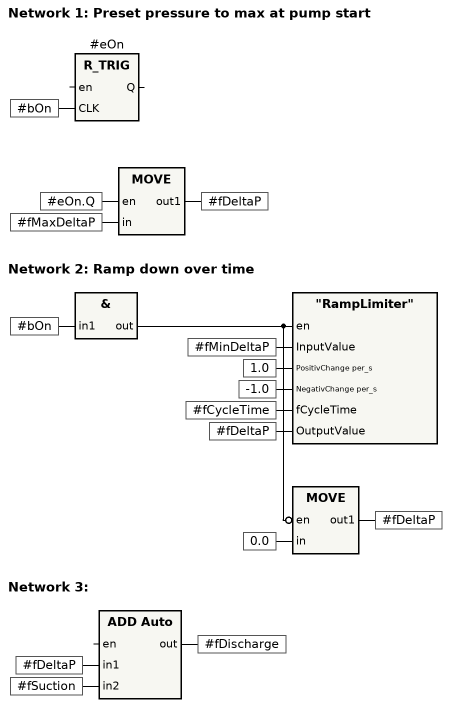
   #eOn(CLK := #bOn);   // R_TRIG
   IF #eOn.Q THEN #fDeltaP := #fMaxDeltaP; END_IF;
END_REGION

REGION Network 2: Ramp down over time
   // When pump is off, delta P is zero.
   // When the pump runs, it starts at the max pressure and ramps down to the min pressure to approximate the decrease in liquid on the suction side
   IF #bOn THEN
       "RampLimiter"(InputValue := #fMinDeltaP,
                     "PositivChange per_s" := 1.0,
                     "NegativChange per_s" := -1.0,
                     fCycleTime := #fCycleTime,
                     OutputValue := #fDeltaP);
   END_IF;
   IF NOT #bOn THEN #fDeltaP := 0.0; END_IF;
END_REGION

REGION Network 3
   #fDischarge := #fDeltaP + #fSuction;
END_REGION
END_FUNCTION_BLOCK

FUNCTION "RampLimiter" : Void
{ S7_Optimized_Access := 'TRUE' }
VERSION : 0.1
   VAR_INPUT 
      InputValue : Real;
      "PositivChange per_s" : Real;
      "NegativChange per_s" : Real;
      fCycleTime : Real;
   END_VAR

   VAR_IN_OUT 
      OutputValue : Real;
   END_VAR


BEGIN
	#OutputValue += MAX(IN1:=MIN(IN1:=#InputValue-#OutputValue,IN2:=#"PositivChange per_s"*#fCycleTime),IN2:=#"NegativChange per_s"*#fCycleTime);
END_FUNCTION

FUNCTION_BLOCK "InputAlarmHandling"   // FB38, FBD
TITLE = Handle I/O alarms
{ S7_Optimized_Access := 'TRUE' }
AUTHOR : Heaten
VERSION : 0.1
// Handle I/O alarms
// stored: AutoNumber true, IsIECCheckEnabled false, IsRetainMemResEnabled false, MemoryReserve 0, SetENOAutomatically false, UDAEnableTagReadback false
   VAR
      A1102 { ExternalAccessible := 'False'; ExternalVisible := 'False'; ExternalWritable := 'False'; S7_SetPoint := 'True'} : "fbDigitalAlarm";
      A1103 { S7_SetPoint := 'True'} : "fbDigitalAlarm";
      A1110 { ExternalAccessible := 'False'; ExternalVisible := 'False'; ExternalWritable := 'False'; S7_SetPoint := 'True'} : "fbDigitalAlarm";
      A1122 { ExternalAccessible := 'False'; ExternalVisible := 'False'; ExternalWritable := 'False'; S7_SetPoint := 'True'} : "fbDigitalAlarm";
      A1123 { S7_SetPoint := 'True'} : "fbDigitalAlarm";
      A1130 { ExternalAccessible := 'False'; ExternalVisible := 'False'; ExternalWritable := 'False'; S7_SetPoint := 'True'} : "fbDigitalAlarm";
      A1142 { ExternalAccessible := 'False'; ExternalVisible := 'False'; ExternalWritable := 'False'; S7_SetPoint := 'True'} : "fbDigitalAlarm";
      A1143 { S7_SetPoint := 'True'} : "fbDigitalAlarm";
      A1150 { ExternalAccessible := 'False'; ExternalVisible := 'False'; ExternalWritable := 'False'; S7_SetPoint := 'True'} : "fbDigitalAlarm";
      A1201 { ExternalAccessible := 'False'; ExternalVisible := 'False'; ExternalWritable := 'False'; S7_SetPoint := 'True'} : "fbHMIEvent";
      A1202 { ExternalAccessible := 'False'; ExternalVisible := 'False'; ExternalWritable := 'False'; S7_SetPoint := 'True'} : "fbHMIEvent";
      A1203 { ExternalAccessible := 'False'; ExternalVisible := 'False'; ExternalWritable := 'False'; S7_SetPoint := 'True'} : "fbHMIEvent";
      A1204 { ExternalAccessible := 'False'; ExternalVisible := 'False'; ExternalWritable := 'False'; S7_SetPoint := 'True'} : "fbHMIEvent";
      A1205 { ExternalAccessible := 'False'; ExternalVisible := 'False'; ExternalWritable := 'False'; S7_SetPoint := 'True'} : "fbHMIEvent";
      A1206 { ExternalAccessible := 'False'; ExternalVisible := 'False'; ExternalWritable := 'False'; S7_SetPoint := 'True'} : "fbHMIEvent";
      A1207 { ExternalAccessible := 'False'; ExternalVisible := 'False'; ExternalWritable := 'False'; S7_SetPoint := 'True'} : "fbHMIEvent";
      A1208 { ExternalAccessible := 'False'; ExternalVisible := 'False'; ExternalWritable := 'False'; S7_SetPoint := 'True'} : "fbHMIEvent";
      A1209 { ExternalAccessible := 'False'; ExternalVisible := 'False'; ExternalWritable := 'False'; S7_SetPoint := 'True'} : "fbHMIEvent";
      A1210 { ExternalAccessible := 'False'; ExternalVisible := 'False'; ExternalWritable := 'False'; S7_SetPoint := 'True'} : "fbHMIEvent";
      A1212 { ExternalAccessible := 'False'; ExternalVisible := 'False'; ExternalWritable := 'False'; S7_SetPoint := 'True'} : "fbHMIEvent";
      A1213 { ExternalAccessible := 'False'; ExternalVisible := 'False'; ExternalWritable := 'False'; S7_SetPoint := 'True'} : "fbHMIEvent";
      A1214 { ExternalAccessible := 'False'; ExternalVisible := 'False'; ExternalWritable := 'False'; S7_SetPoint := 'True'} : "fbHMIEvent";
      A1215 { ExternalAccessible := 'False'; ExternalVisible := 'False'; ExternalWritable := 'False'; S7_SetPoint := 'True'} : "fbHMIEvent";
      A1220 { ExternalAccessible := 'False'; ExternalVisible := 'False'; ExternalWritable := 'False'; S7_SetPoint := 'True'} : "fbHMIEvent";
      A1221 { ExternalAccessible := 'False'; ExternalVisible := 'False'; ExternalWritable := 'False'; S7_SetPoint := 'True'} : "fbHMIEvent";
      A1223 { ExternalAccessible := 'False'; ExternalVisible := 'False'; ExternalWritable := 'False'; S7_SetPoint := 'True'} : "fbHMIEvent";
      A1231 { ExternalAccessible := 'False'; ExternalVisible := 'False'; ExternalWritable := 'False'; S7_SetPoint := 'True'} : "fbHMIEvent";
      A1232 { ExternalAccessible := 'False'; ExternalVisible := 'False'; ExternalWritable := 'False'; S7_SetPoint := 'True'} : "fbHMIEvent";
      A1233 { ExternalAccessible := 'False'; ExternalVisible := 'False'; ExternalWritable := 'False'; S7_SetPoint := 'True'} : "fbDigitalAlarm";
      A1241 { ExternalAccessible := 'False'; ExternalVisible := 'False'; ExternalWritable := 'False'; S7_SetPoint := 'True'} : "fbHMIEvent";
      A1242 { ExternalAccessible := 'False'; ExternalVisible := 'False'; ExternalWritable := 'False'; S7_SetPoint := 'True'} : "fbHMIEvent";
      A1243 { ExternalAccessible := 'False'; ExternalVisible := 'False'; ExternalWritable := 'False'; S7_SetPoint := 'True'} : "fbHMIEvent";
      A1244 { ExternalAccessible := 'False'; ExternalVisible := 'False'; ExternalWritable := 'False'; S7_SetPoint := 'True'} : "fbHMIEvent";
      A1255 { ExternalAccessible := 'False'; ExternalVisible := 'False'; ExternalWritable := 'False'; S7_SetPoint := 'True'} : "fbHMIEvent";
      A1256 { ExternalAccessible := 'False'; ExternalVisible := 'False'; ExternalWritable := 'False'; S7_SetPoint := 'True'} : "fbHMIEvent";
      A1257 { ExternalAccessible := 'False'; ExternalVisible := 'False'; ExternalWritable := 'False'; S7_SetPoint := 'True'} : "fbHMIEvent";
      A1264 { ExternalAccessible := 'False'; ExternalVisible := 'False'; ExternalWritable := 'False'; S7_SetPoint := 'True'} : "fbHMIEvent";
      A1266 { ExternalAccessible := 'False'; ExternalVisible := 'False'; ExternalWritable := 'False'; S7_SetPoint := 'True'} : "fbHMIEvent";
      A1267 { ExternalAccessible := 'False'; ExternalVisible := 'False'; ExternalWritable := 'False'; S7_SetPoint := 'True'} : "fbHMIEvent";
      A1268 { ExternalAccessible := 'False'; ExternalVisible := 'False'; ExternalWritable := 'False'; S7_SetPoint := 'True'} : "fbHMIEvent";
      A1274 { S7_SetPoint := 'True'} : "fbHMIEvent";
      A1276 { S7_SetPoint := 'True'} : "fbHMIEvent";
      A1277 { S7_SetPoint := 'True'} : "fbHMIEvent";
      A1278 { S7_SetPoint := 'True'} : "fbHMIEvent";
      A1279 { S7_SetPoint := 'True'} : "fbHMIEvent";
      A1280 { S7_SetPoint := 'True'} : "fbHMIEvent";
      A1281 { S7_SetPoint := 'True'} : "fbHMIEvent";
      A1282 { S7_SetPoint := 'True'} : "fbHMIEvent";
      A1283 { S7_SetPoint := 'True'} : "fbHMIEvent";
      A1284 { S7_SetPoint := 'True'} : "fbHMIEvent";
      A1285 { S7_SetPoint := 'True'} : "fbHMIEvent";
      A1286 { S7_SetPoint := 'True'} : "fbHMIEvent";
      A1287 { S7_SetPoint := 'True'} : "fbHMIEvent";
      A1288 { S7_SetPoint := 'True'} : "fbHMIEvent";
      A1289 { S7_SetPoint := 'True'} : "fbHMIEvent";
      A1290 { S7_SetPoint := 'True'} : "fbHMIEvent";
      A1291 { S7_SetPoint := 'True'} : "fbHMIEvent";
      A1292 { S7_SetPoint := 'True'} : "fbHMIEvent";
      A5250 { ExternalAccessible := 'False'; ExternalVisible := 'False'; ExternalWritable := 'False'; S7_SetPoint := 'True'} : "fbHMIEvent";
      A5251 { ExternalAccessible := 'False'; ExternalVisible := 'False'; ExternalWritable := 'False'; S7_SetPoint := 'True'} : "fbHMIEvent";
      A5252 { ExternalAccessible := 'False'; ExternalVisible := 'False'; ExternalWritable := 'False'; S7_SetPoint := 'True'} : "fbHMIEvent";
      A5253 { ExternalAccessible := 'False'; ExternalVisible := 'False'; ExternalWritable := 'False'; S7_SetPoint := 'True'} : "fbHMIEvent";
      A5254 { ExternalAccessible := 'False'; ExternalVisible := 'False'; ExternalWritable := 'False'; S7_SetPoint := 'True'} : "fbHMIEvent";
      A5255 { ExternalAccessible := 'False'; ExternalVisible := 'False'; ExternalWritable := 'False'; S7_SetPoint := 'True'} : "fbHMIEvent";
   END_VAR
BEGIN

REGION Network 1: 1102
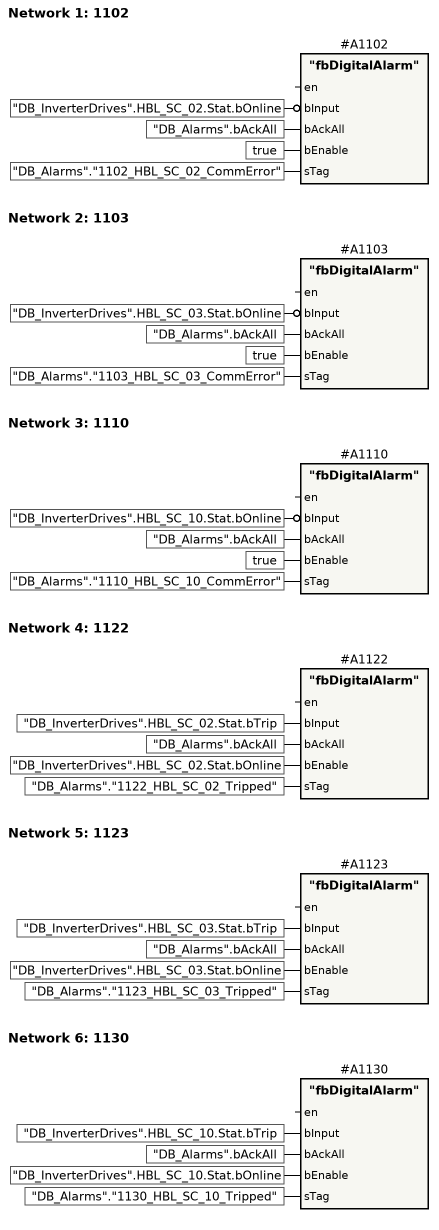
   #A1102(bInput := NOT "DB_InverterDrives".HBL_SC_02.Stat.bOnline,   // "fbDigitalAlarm"
          bAckAll := "DB_Alarms".bAckAll,
          bEnable := true,
          sTag := "DB_Alarms"."1102_HBL_SC_02_CommError");
END_REGION

REGION Network 2: 1103
   #A1103(bInput := NOT "DB_InverterDrives".HBL_SC_03.Stat.bOnline,   // "fbDigitalAlarm"
          bAckAll := "DB_Alarms".bAckAll,
          bEnable := true,
          sTag := "DB_Alarms"."1103_HBL_SC_03_CommError");
END_REGION

REGION Network 3: 1110
   #A1110(bInput := NOT "DB_InverterDrives".HBL_SC_10.Stat.bOnline,   // "fbDigitalAlarm"
          bAckAll := "DB_Alarms".bAckAll,
          bEnable := true,
          sTag := "DB_Alarms"."1110_HBL_SC_10_CommError");
END_REGION

REGION Network 4: 1122
   // Only show if online
   #A1122(bInput := "DB_InverterDrives".HBL_SC_02.Stat.bTrip,   // "fbDigitalAlarm"
          bAckAll := "DB_Alarms".bAckAll,
          bEnable := "DB_InverterDrives".HBL_SC_02.Stat.bOnline,
          sTag := "DB_Alarms"."1122_HBL_SC_02_Tripped");
END_REGION

REGION Network 5: 1123
   // Only show if online
   #A1123(bInput := "DB_InverterDrives".HBL_SC_03.Stat.bTrip,   // "fbDigitalAlarm"
          bAckAll := "DB_Alarms".bAckAll,
          bEnable := "DB_InverterDrives".HBL_SC_03.Stat.bOnline,
          sTag := "DB_Alarms"."1123_HBL_SC_03_Tripped");
END_REGION

REGION Network 6: 1130
   // Only show if online
   #A1130(bInput := "DB_InverterDrives".HBL_SC_10.Stat.bTrip,   // "fbDigitalAlarm"
          bAckAll := "DB_Alarms".bAckAll,
          bEnable := "DB_InverterDrives".HBL_SC_10.Stat.bOnline,
          sTag := "DB_Alarms"."1130_HBL_SC_10_Tripped");
END_REGION

REGION Network 7: 1142
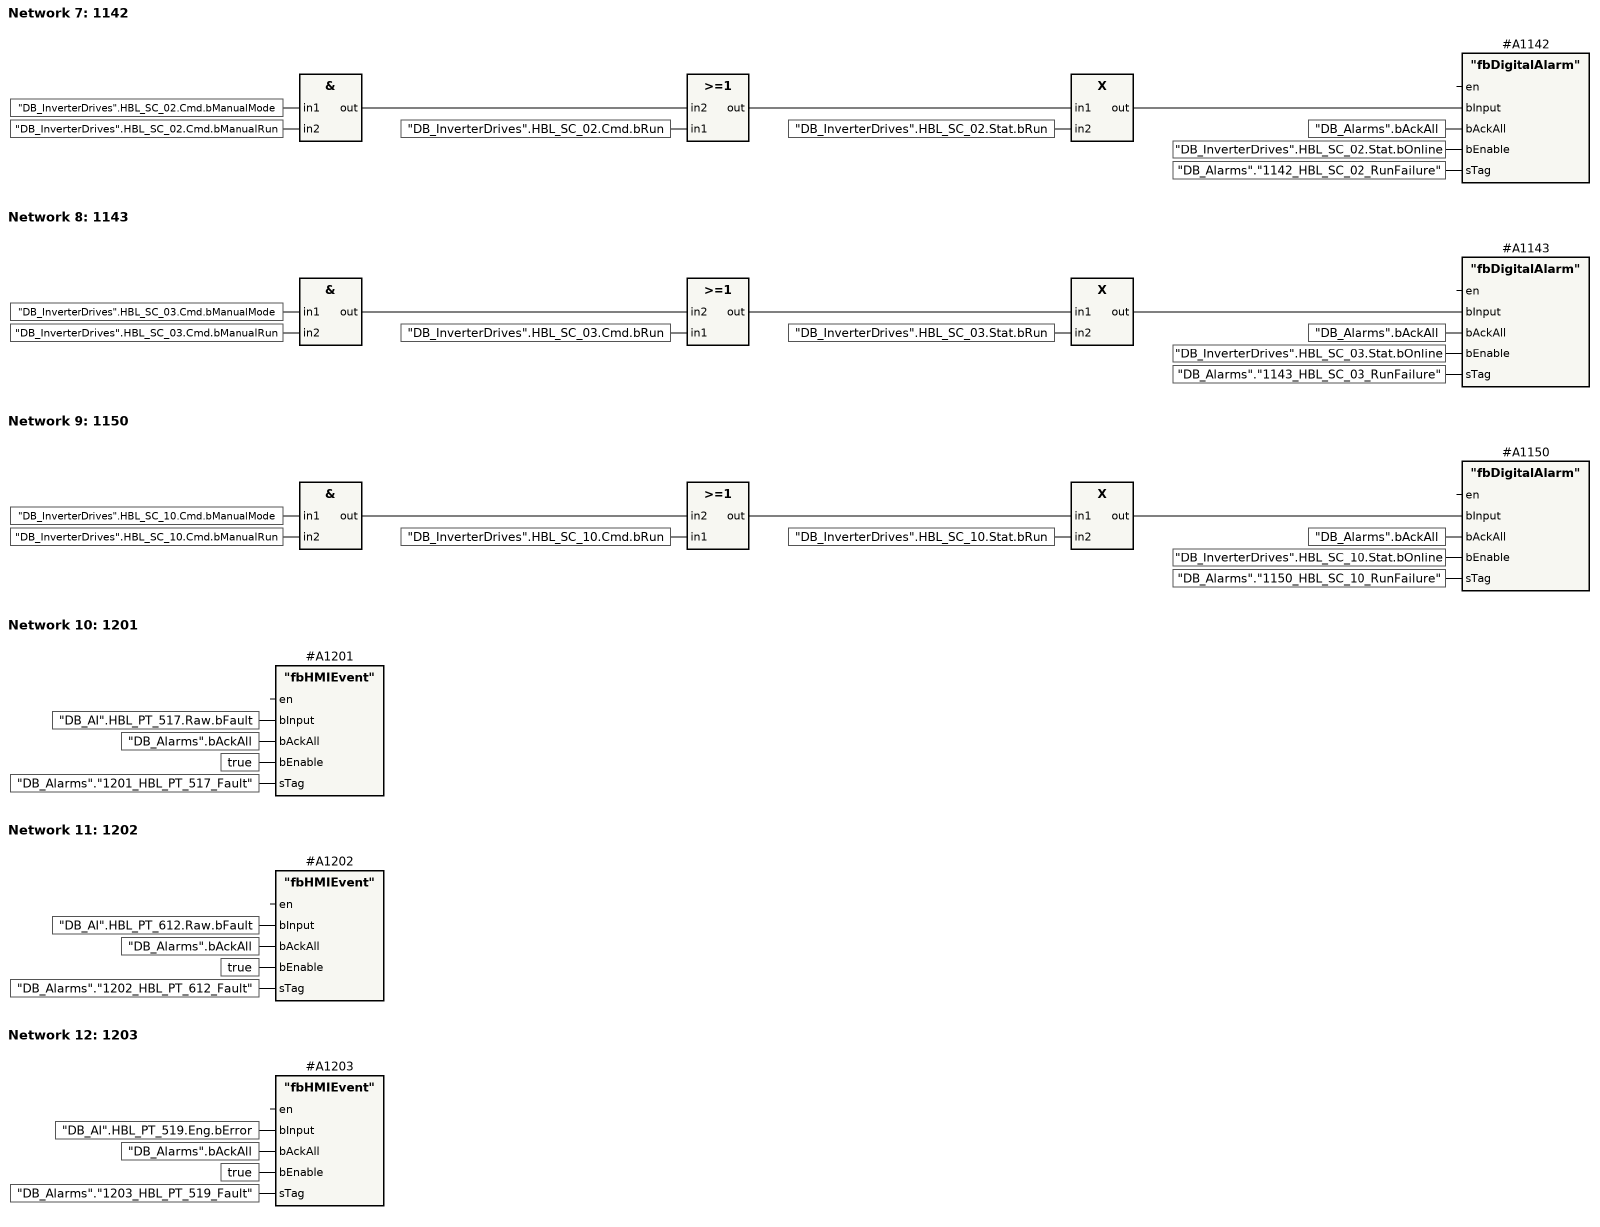
   #A1142(bInput := (("DB_InverterDrives".HBL_SC_02.Cmd.bManualMode AND "DB_InverterDrives".HBL_SC_02.Cmd.bManualRun) OR "DB_InverterDrives".HBL_SC_02.Cmd.bRun) XOR "DB_InverterDrives".HBL_SC_02.Stat.bRun,   // "fbDigitalAlarm"
          bAckAll := "DB_Alarms".bAckAll,
          bEnable := "DB_InverterDrives".HBL_SC_02.Stat.bOnline,
          sTag := "DB_Alarms"."1142_HBL_SC_02_RunFailure");
END_REGION

REGION Network 8: 1143
   #A1143(bInput := (("DB_InverterDrives".HBL_SC_03.Cmd.bManualMode AND "DB_InverterDrives".HBL_SC_03.Cmd.bManualRun) OR "DB_InverterDrives".HBL_SC_03.Cmd.bRun) XOR "DB_InverterDrives".HBL_SC_03.Stat.bRun,   // "fbDigitalAlarm"
          bAckAll := "DB_Alarms".bAckAll,
          bEnable := "DB_InverterDrives".HBL_SC_03.Stat.bOnline,
          sTag := "DB_Alarms"."1143_HBL_SC_03_RunFailure");
END_REGION

REGION Network 9: 1150
   #A1150(bInput := (("DB_InverterDrives".HBL_SC_10.Cmd.bManualMode AND "DB_InverterDrives".HBL_SC_10.Cmd.bManualRun) OR "DB_InverterDrives".HBL_SC_10.Cmd.bRun) XOR "DB_InverterDrives".HBL_SC_10.Stat.bRun,   // "fbDigitalAlarm"
          bAckAll := "DB_Alarms".bAckAll,
          bEnable := "DB_InverterDrives".HBL_SC_10.Stat.bOnline,
          sTag := "DB_Alarms"."1150_HBL_SC_10_RunFailure");
END_REGION

REGION Network 10: 1201
   #A1201(bInput := "DB_AI".HBL_PT_517.Raw.bFault,   // "fbHMIEvent"
          bAckAll := "DB_Alarms".bAckAll,
          bEnable := true,
          sTag := "DB_Alarms"."1201_HBL_PT_517_Fault");
END_REGION

REGION Network 11: 1202
   #A1202(bInput := "DB_AI".HBL_PT_612.Raw.bFault,   // "fbHMIEvent"
          bAckAll := "DB_Alarms".bAckAll,
          bEnable := true,
          sTag := "DB_Alarms"."1202_HBL_PT_612_Fault");
END_REGION

REGION Network 12: 1203
   #A1203(bInput := "DB_AI".HBL_PT_519.Eng.bError,   // "fbHMIEvent"
          bAckAll := "DB_Alarms".bAckAll,
          bEnable := true,
          sTag := "DB_Alarms"."1203_HBL_PT_519_Fault");
END_REGION

REGION Network 13: 1204
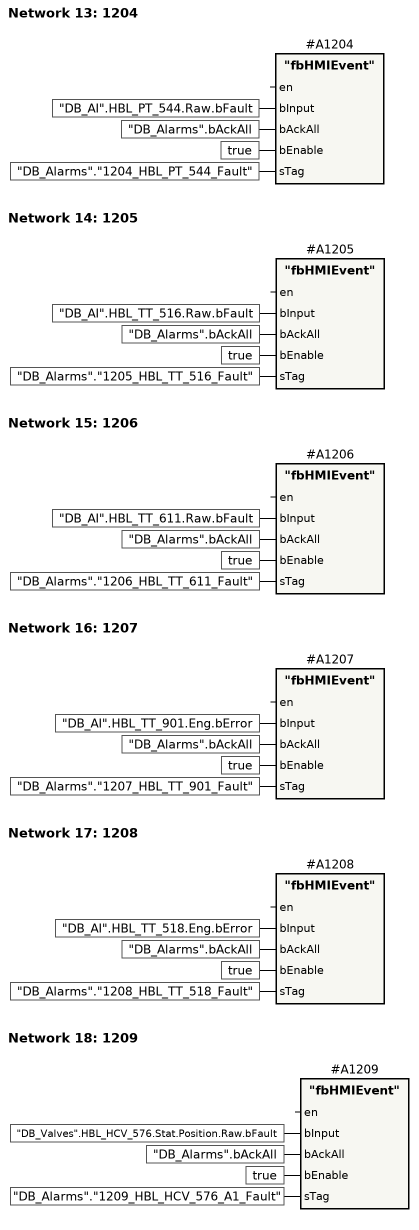
   #A1204(bInput := "DB_AI".HBL_PT_544.Raw.bFault,   // "fbHMIEvent"
          bAckAll := "DB_Alarms".bAckAll,
          bEnable := true,
          sTag := "DB_Alarms"."1204_HBL_PT_544_Fault");
END_REGION

REGION Network 14: 1205
   #A1205(bInput := "DB_AI".HBL_TT_516.Raw.bFault,   // "fbHMIEvent"
          bAckAll := "DB_Alarms".bAckAll,
          bEnable := true,
          sTag := "DB_Alarms"."1205_HBL_TT_516_Fault");
END_REGION

REGION Network 15: 1206
   #A1206(bInput := "DB_AI".HBL_TT_611.Raw.bFault,   // "fbHMIEvent"
          bAckAll := "DB_Alarms".bAckAll,
          bEnable := true,
          sTag := "DB_Alarms"."1206_HBL_TT_611_Fault");
END_REGION

REGION Network 16: 1207
   #A1207(bInput := "DB_AI".HBL_TT_901.Eng.bError,   // "fbHMIEvent"
          bAckAll := "DB_Alarms".bAckAll,
          bEnable := true,
          sTag := "DB_Alarms"."1207_HBL_TT_901_Fault");
END_REGION

REGION Network 17: 1208
   #A1208(bInput := "DB_AI".HBL_TT_518.Eng.bError,   // "fbHMIEvent"
          bAckAll := "DB_Alarms".bAckAll,
          bEnable := true,
          sTag := "DB_Alarms"."1208_HBL_TT_518_Fault");
END_REGION

REGION Network 18: 1209
   #A1209(bInput := "DB_Valves".HBL_HCV_576.Stat.Position.Raw.bFault,   // "fbHMIEvent"
          bAckAll := "DB_Alarms".bAckAll,
          bEnable := true,
          sTag := "DB_Alarms"."1209_HBL_HCV_576_A1_Fault");
END_REGION

REGION Network 19: 1210
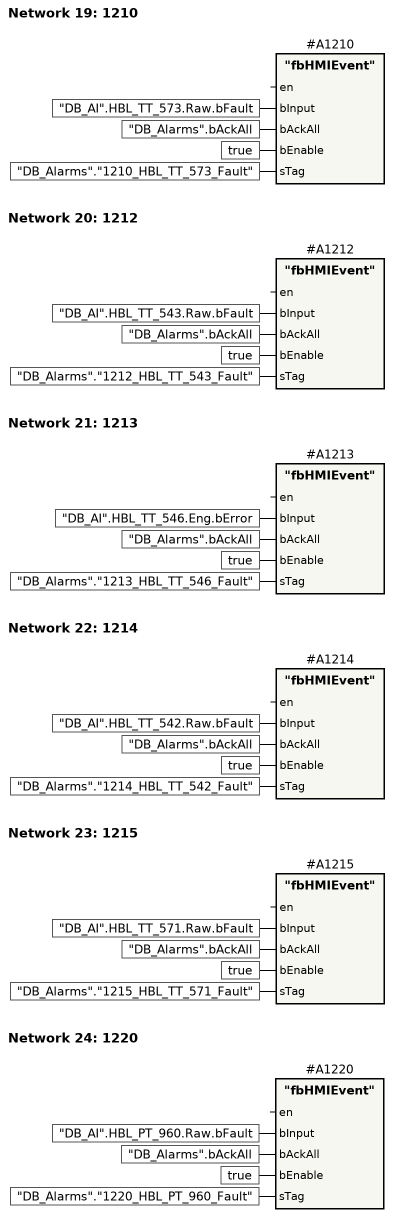
   #A1210(bInput := "DB_AI".HBL_TT_573.Raw.bFault,   // "fbHMIEvent"
          bAckAll := "DB_Alarms".bAckAll,
          bEnable := true,
          sTag := "DB_Alarms"."1210_HBL_TT_573_Fault");
END_REGION

REGION Network 20: 1212
   #A1212(bInput := "DB_AI".HBL_TT_543.Raw.bFault,   // "fbHMIEvent"
          bAckAll := "DB_Alarms".bAckAll,
          bEnable := true,
          sTag := "DB_Alarms"."1212_HBL_TT_543_Fault");
END_REGION

REGION Network 21: 1213
   #A1213(bInput := "DB_AI".HBL_TT_546.Eng.bError,   // "fbHMIEvent"
          bAckAll := "DB_Alarms".bAckAll,
          bEnable := true,
          sTag := "DB_Alarms"."1213_HBL_TT_546_Fault");
END_REGION

REGION Network 22: 1214
   #A1214(bInput := "DB_AI".HBL_TT_542.Raw.bFault,   // "fbHMIEvent"
          bAckAll := "DB_Alarms".bAckAll,
          bEnable := true,
          sTag := "DB_Alarms"."1214_HBL_TT_542_Fault");
END_REGION

REGION Network 23: 1215
   #A1215(bInput := "DB_AI".HBL_TT_571.Raw.bFault,   // "fbHMIEvent"
          bAckAll := "DB_Alarms".bAckAll,
          bEnable := true,
          sTag := "DB_Alarms"."1215_HBL_TT_571_Fault");
END_REGION

REGION Network 24: 1220
   #A1220(bInput := "DB_AI".HBL_PT_960.Raw.bFault,   // "fbHMIEvent"
          bAckAll := "DB_Alarms".bAckAll,
          bEnable := true,
          sTag := "DB_Alarms"."1220_HBL_PT_960_Fault");
END_REGION

REGION Network 25: 1221
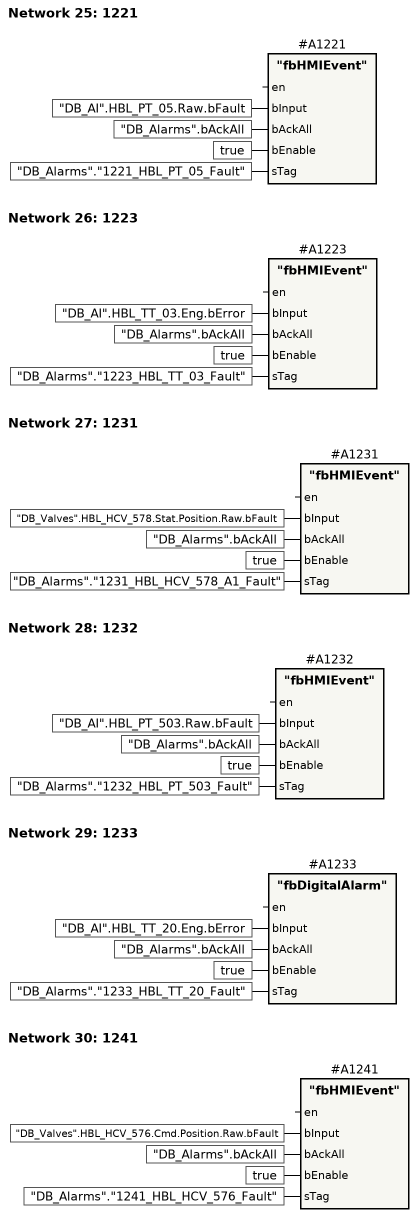
   #A1221(bInput := "DB_AI".HBL_PT_05.Raw.bFault,   // "fbHMIEvent"
          bAckAll := "DB_Alarms".bAckAll,
          bEnable := true,
          sTag := "DB_Alarms"."1221_HBL_PT_05_Fault");
END_REGION

REGION Network 26: 1223
   #A1223(bInput := "DB_AI".HBL_TT_03.Eng.bError,   // "fbHMIEvent"
          bAckAll := "DB_Alarms".bAckAll,
          bEnable := true,
          sTag := "DB_Alarms"."1223_HBL_TT_03_Fault");
END_REGION

REGION Network 27: 1231
   #A1231(bInput := "DB_Valves".HBL_HCV_578.Stat.Position.Raw.bFault,   // "fbHMIEvent"
          bAckAll := "DB_Alarms".bAckAll,
          bEnable := true,
          sTag := "DB_Alarms"."1231_HBL_HCV_578_A1_Fault");
END_REGION

REGION Network 28: 1232
   #A1232(bInput := "DB_AI".HBL_PT_503.Raw.bFault,   // "fbHMIEvent"
          bAckAll := "DB_Alarms".bAckAll,
          bEnable := true,
          sTag := "DB_Alarms"."1232_HBL_PT_503_Fault");
END_REGION

REGION Network 29: 1233
   #A1233(bInput := "DB_AI".HBL_TT_20.Eng.bError,   // "fbDigitalAlarm"
          bAckAll := "DB_Alarms".bAckAll,
          bEnable := true,
          sTag := "DB_Alarms"."1233_HBL_TT_20_Fault");
END_REGION

REGION Network 30: 1241
   #A1241(bInput := "DB_Valves".HBL_HCV_576.Cmd.Position.Raw.bFault,   // "fbHMIEvent"
          bAckAll := "DB_Alarms".bAckAll,
          bEnable := true,
          sTag := "DB_Alarms"."1241_HBL_HCV_576_Fault");
END_REGION

REGION Network 31: 1242
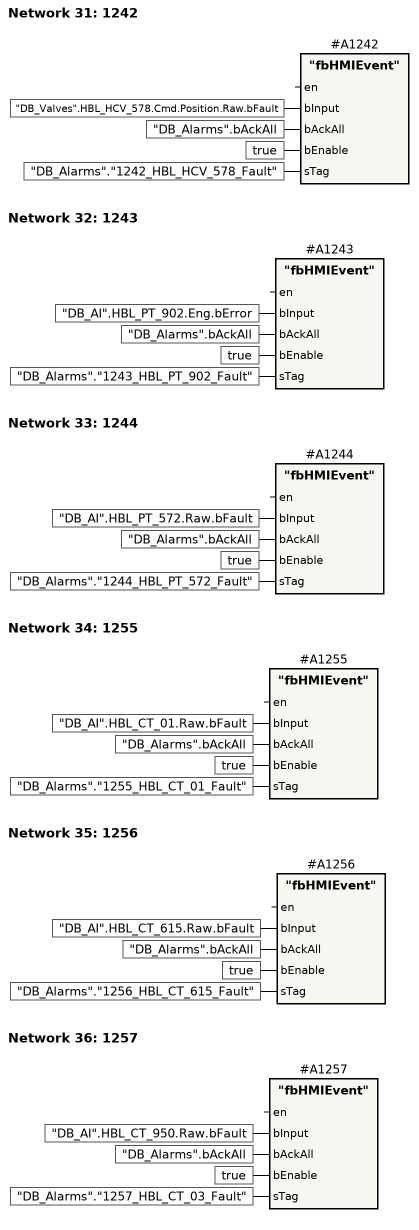
   #A1242(bInput := "DB_Valves".HBL_HCV_578.Cmd.Position.Raw.bFault,   // "fbHMIEvent"
          bAckAll := "DB_Alarms".bAckAll,
          bEnable := true,
          sTag := "DB_Alarms"."1242_HBL_HCV_578_Fault");
END_REGION

REGION Network 32: 1243
   #A1243(bInput := "DB_AI".HBL_PT_902.Eng.bError,   // "fbHMIEvent"
          bAckAll := "DB_Alarms".bAckAll,
          bEnable := true,
          sTag := "DB_Alarms"."1243_HBL_PT_902_Fault");
END_REGION

REGION Network 33: 1244
   #A1244(bInput := "DB_AI".HBL_PT_572.Raw.bFault,   // "fbHMIEvent"
          bAckAll := "DB_Alarms".bAckAll,
          bEnable := true,
          sTag := "DB_Alarms"."1244_HBL_PT_572_Fault");
END_REGION

REGION Network 34: 1255
   #A1255(bInput := "DB_AI".HBL_CT_01.Raw.bFault,   // "fbHMIEvent"
          bAckAll := "DB_Alarms".bAckAll,
          bEnable := true,
          sTag := "DB_Alarms"."1255_HBL_CT_01_Fault");
END_REGION

REGION Network 35: 1256
   #A1256(bInput := "DB_AI".HBL_CT_615.Raw.bFault,   // "fbHMIEvent"
          bAckAll := "DB_Alarms".bAckAll,
          bEnable := true,
          sTag := "DB_Alarms"."1256_HBL_CT_615_Fault");
END_REGION

REGION Network 36: 1257
   #A1257(bInput := "DB_AI".HBL_CT_950.Raw.bFault,   // "fbHMIEvent"
          bAckAll := "DB_Alarms".bAckAll,
          bEnable := true,
          sTag := "DB_Alarms"."1257_HBL_CT_03_Fault");
END_REGION

REGION Network 37: 1264
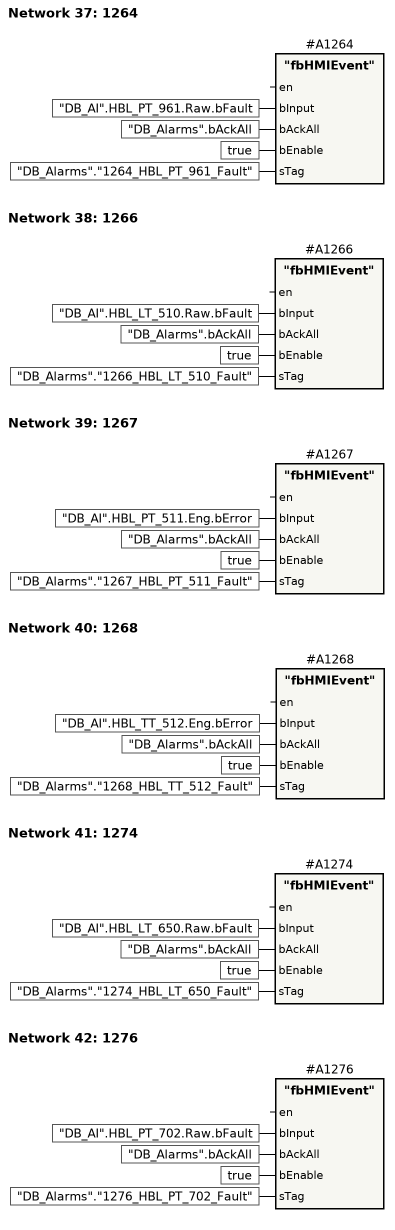
   #A1264(bInput := "DB_AI".HBL_PT_961.Raw.bFault,   // "fbHMIEvent"
          bAckAll := "DB_Alarms".bAckAll,
          bEnable := true,
          sTag := "DB_Alarms"."1264_HBL_PT_961_Fault");
END_REGION

REGION Network 38: 1266
   #A1266(bInput := "DB_AI".HBL_LT_510.Raw.bFault,   // "fbHMIEvent"
          bAckAll := "DB_Alarms".bAckAll,
          bEnable := true,
          sTag := "DB_Alarms"."1266_HBL_LT_510_Fault");
END_REGION

REGION Network 39: 1267
   #A1267(bInput := "DB_AI".HBL_PT_511.Eng.bError,   // "fbHMIEvent"
          bAckAll := "DB_Alarms".bAckAll,
          bEnable := true,
          sTag := "DB_Alarms"."1267_HBL_PT_511_Fault");
END_REGION

REGION Network 40: 1268
   #A1268(bInput := "DB_AI".HBL_TT_512.Eng.bError,   // "fbHMIEvent"
          bAckAll := "DB_Alarms".bAckAll,
          bEnable := true,
          sTag := "DB_Alarms"."1268_HBL_TT_512_Fault");
END_REGION

REGION Network 41: 1274
   #A1274(bInput := "DB_AI".HBL_LT_650.Raw.bFault,   // "fbHMIEvent"
          bAckAll := "DB_Alarms".bAckAll,
          bEnable := true,
          sTag := "DB_Alarms"."1274_HBL_LT_650_Fault");
END_REGION

REGION Network 42: 1276
   #A1276(bInput := "DB_AI".HBL_PT_702.Raw.bFault,   // "fbHMIEvent"
          bAckAll := "DB_Alarms".bAckAll,
          bEnable := true,
          sTag := "DB_Alarms"."1276_HBL_PT_702_Fault");
END_REGION

REGION Network 43: 1277
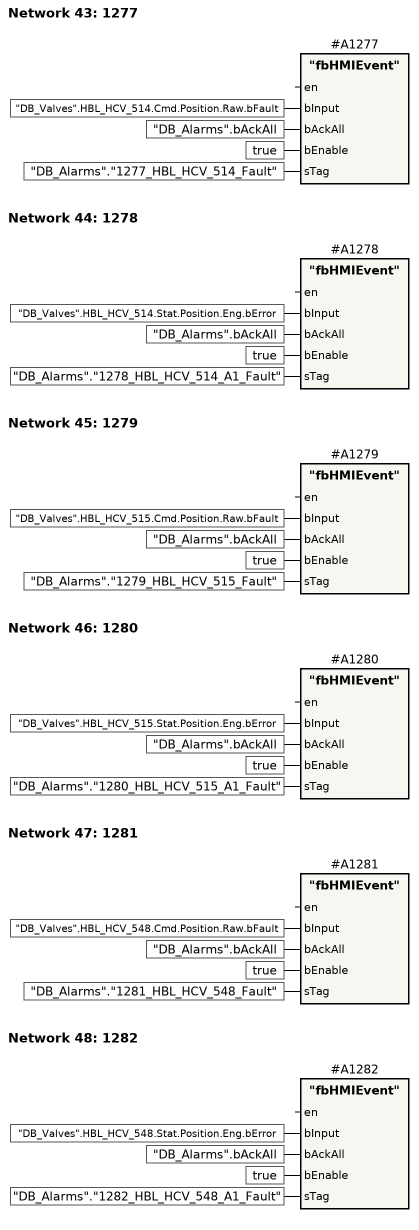
   #A1277(bInput := "DB_Valves".HBL_HCV_514.Cmd.Position.Raw.bFault,   // "fbHMIEvent"
          bAckAll := "DB_Alarms".bAckAll,
          bEnable := true,
          sTag := "DB_Alarms"."1277_HBL_HCV_514_Fault");
END_REGION

REGION Network 44: 1278
   #A1278(bInput := "DB_Valves".HBL_HCV_514.Stat.Position.Eng.bError,   // "fbHMIEvent"
          bAckAll := "DB_Alarms".bAckAll,
          bEnable := true,
          sTag := "DB_Alarms"."1278_HBL_HCV_514_A1_Fault");
END_REGION

REGION Network 45: 1279
   #A1279(bInput := "DB_Valves".HBL_HCV_515.Cmd.Position.Raw.bFault,   // "fbHMIEvent"
          bAckAll := "DB_Alarms".bAckAll,
          bEnable := true,
          sTag := "DB_Alarms"."1279_HBL_HCV_515_Fault");
END_REGION

REGION Network 46: 1280
   #A1280(bInput := "DB_Valves".HBL_HCV_515.Stat.Position.Eng.bError,   // "fbHMIEvent"
          bAckAll := "DB_Alarms".bAckAll,
          bEnable := true,
          sTag := "DB_Alarms"."1280_HBL_HCV_515_A1_Fault");
END_REGION

REGION Network 47: 1281
   #A1281(bInput := "DB_Valves".HBL_HCV_548.Cmd.Position.Raw.bFault,   // "fbHMIEvent"
          bAckAll := "DB_Alarms".bAckAll,
          bEnable := true,
          sTag := "DB_Alarms"."1281_HBL_HCV_548_Fault");
END_REGION

REGION Network 48: 1282
   #A1282(bInput := "DB_Valves".HBL_HCV_548.Stat.Position.Eng.bError,   // "fbHMIEvent"
          bAckAll := "DB_Alarms".bAckAll,
          bEnable := true,
          sTag := "DB_Alarms"."1282_HBL_HCV_548_A1_Fault");
END_REGION

REGION Network 49: 1283
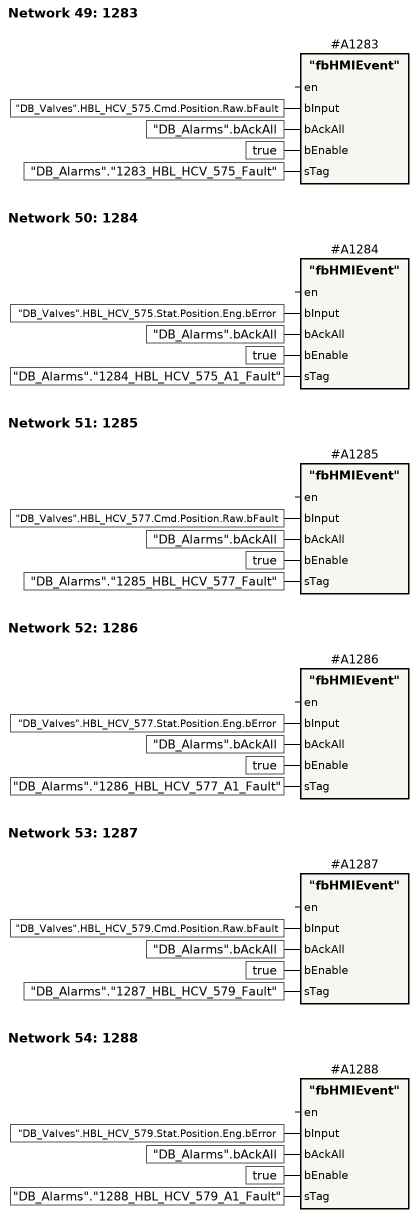
   #A1283(bInput := "DB_Valves".HBL_HCV_575.Cmd.Position.Raw.bFault,   // "fbHMIEvent"
          bAckAll := "DB_Alarms".bAckAll,
          bEnable := true,
          sTag := "DB_Alarms"."1283_HBL_HCV_575_Fault");
END_REGION

REGION Network 50: 1284
   #A1284(bInput := "DB_Valves".HBL_HCV_575.Stat.Position.Eng.bError,   // "fbHMIEvent"
          bAckAll := "DB_Alarms".bAckAll,
          bEnable := true,
          sTag := "DB_Alarms"."1284_HBL_HCV_575_A1_Fault");
END_REGION

REGION Network 51: 1285
   #A1285(bInput := "DB_Valves".HBL_HCV_577.Cmd.Position.Raw.bFault,   // "fbHMIEvent"
          bAckAll := "DB_Alarms".bAckAll,
          bEnable := true,
          sTag := "DB_Alarms"."1285_HBL_HCV_577_Fault");
END_REGION

REGION Network 52: 1286
   #A1286(bInput := "DB_Valves".HBL_HCV_577.Stat.Position.Eng.bError,   // "fbHMIEvent"
          bAckAll := "DB_Alarms".bAckAll,
          bEnable := true,
          sTag := "DB_Alarms"."1286_HBL_HCV_577_A1_Fault");
END_REGION

REGION Network 53: 1287
   #A1287(bInput := "DB_Valves".HBL_HCV_579.Cmd.Position.Raw.bFault,   // "fbHMIEvent"
          bAckAll := "DB_Alarms".bAckAll,
          bEnable := true,
          sTag := "DB_Alarms"."1287_HBL_HCV_579_Fault");
END_REGION

REGION Network 54: 1288
   #A1288(bInput := "DB_Valves".HBL_HCV_579.Stat.Position.Eng.bError,   // "fbHMIEvent"
          bAckAll := "DB_Alarms".bAckAll,
          bEnable := true,
          sTag := "DB_Alarms"."1288_HBL_HCV_579_A1_Fault");
END_REGION

REGION Network 55: 1289
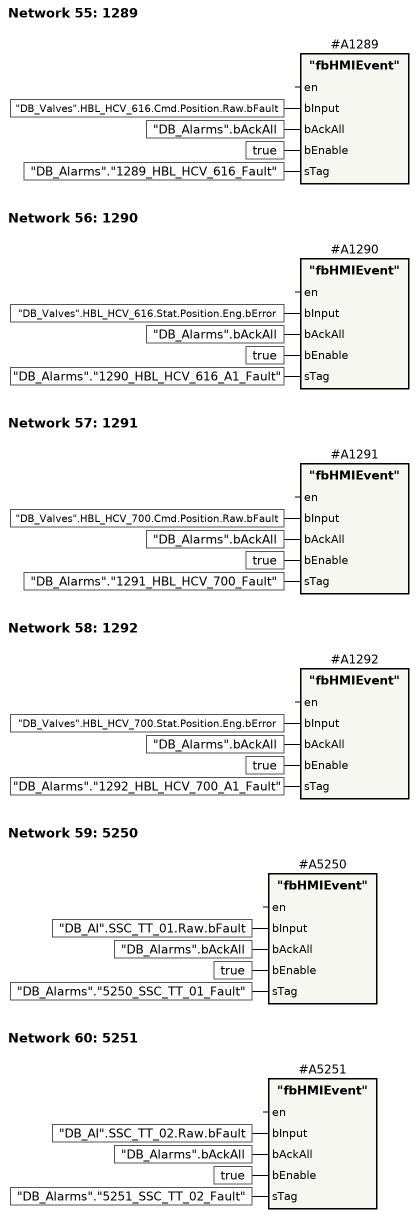
   #A1289(bInput := "DB_Valves".HBL_HCV_616.Cmd.Position.Raw.bFault,   // "fbHMIEvent"
          bAckAll := "DB_Alarms".bAckAll,
          bEnable := true,
          sTag := "DB_Alarms"."1289_HBL_HCV_616_Fault");
END_REGION

REGION Network 56: 1290
   #A1290(bInput := "DB_Valves".HBL_HCV_616.Stat.Position.Eng.bError,   // "fbHMIEvent"
          bAckAll := "DB_Alarms".bAckAll,
          bEnable := true,
          sTag := "DB_Alarms"."1290_HBL_HCV_616_A1_Fault");
END_REGION

REGION Network 57: 1291
   #A1291(bInput := "DB_Valves".HBL_HCV_700.Cmd.Position.Raw.bFault,   // "fbHMIEvent"
          bAckAll := "DB_Alarms".bAckAll,
          bEnable := true,
          sTag := "DB_Alarms"."1291_HBL_HCV_700_Fault");
END_REGION

REGION Network 58: 1292
   #A1292(bInput := "DB_Valves".HBL_HCV_700.Stat.Position.Eng.bError,   // "fbHMIEvent"
          bAckAll := "DB_Alarms".bAckAll,
          bEnable := true,
          sTag := "DB_Alarms"."1292_HBL_HCV_700_A1_Fault");
END_REGION

REGION Network 59: 5250
   #A5250(bInput := "DB_AI".SSC_TT_01.Raw.bFault,   // "fbHMIEvent"
          bAckAll := "DB_Alarms".bAckAll,
          bEnable := true,
          sTag := "DB_Alarms"."5250_SSC_TT_01_Fault");
END_REGION

REGION Network 60: 5251
   #A5251(bInput := "DB_AI".SSC_TT_02.Raw.bFault,   // "fbHMIEvent"
          bAckAll := "DB_Alarms".bAckAll,
          bEnable := true,
          sTag := "DB_Alarms"."5251_SSC_TT_02_Fault");
END_REGION

REGION Network 61: 5252
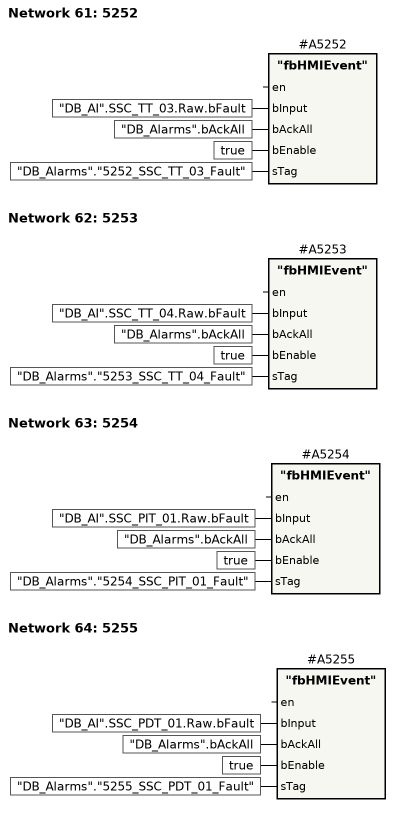
   #A5252(bInput := "DB_AI".SSC_TT_03.Raw.bFault,   // "fbHMIEvent"
          bAckAll := "DB_Alarms".bAckAll,
          bEnable := true,
          sTag := "DB_Alarms"."5252_SSC_TT_03_Fault");
END_REGION

REGION Network 62: 5253
   #A5253(bInput := "DB_AI".SSC_TT_04.Raw.bFault,   // "fbHMIEvent"
          bAckAll := "DB_Alarms".bAckAll,
          bEnable := true,
          sTag := "DB_Alarms"."5253_SSC_TT_04_Fault");
END_REGION

REGION Network 63: 5254
   #A5254(bInput := "DB_AI".SSC_PIT_01.Raw.bFault,   // "fbHMIEvent"
          bAckAll := "DB_Alarms".bAckAll,
          bEnable := true,
          sTag := "DB_Alarms"."5254_SSC_PIT_01_Fault");
END_REGION

REGION Network 64: 5255
   #A5255(bInput := "DB_AI".SSC_PDT_01.Raw.bFault,   // "fbHMIEvent"
          bAckAll := "DB_Alarms".bAckAll,
          bEnable := true,
          sTag := "DB_Alarms"."5255_SSC_PDT_01_Fault");
END_REGION
END_FUNCTION_BLOCK

FUNCTION "Control" : Void   // FC3, FBD
TITLE = Sequencing of control algorithms
{ S7_Optimized_Access := 'TRUE' }
AUTHOR : Heaten
VERSION : 0.1
// stored: AutoNumber true, IsIECCheckEnabled false, SetENOAutomatically false, UDAEnableTagReadback false
BEGIN

REGION Network 1: Calculations for process controlling and monitoring
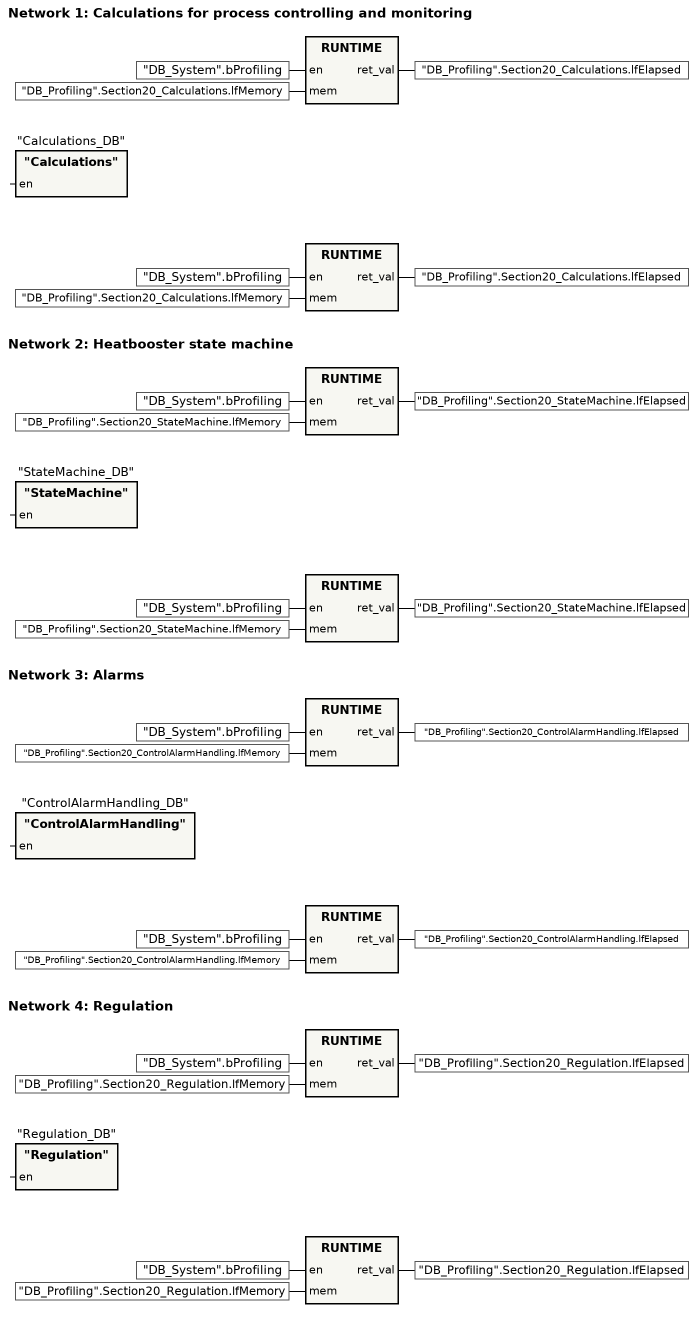
   // no SCL statement known for Runtime: written as a call
   IF "DB_System".bProfiling THEN
       "DB_Profiling".Section20_Calculations.lfElapsed := Runtime(mem := "DB_Profiling".Section20_Calculations.lfMemory);
   END_IF;
   "Calculations_DB"();   // "Calculations"
   IF "DB_System".bProfiling THEN
       "DB_Profiling".Section20_Calculations.lfElapsed := Runtime(mem := "DB_Profiling".Section20_Calculations.lfMemory);
   END_IF;
END_REGION

REGION Network 2: Heatbooster state machine
   // no SCL statement known for Runtime: written as a call
   IF "DB_System".bProfiling THEN
       "DB_Profiling".Section20_StateMachine.lfElapsed := Runtime(mem := "DB_Profiling".Section20_StateMachine.lfMemory);
   END_IF;
   "StateMachine_DB"();   // "StateMachine"
   IF "DB_System".bProfiling THEN
       "DB_Profiling".Section20_StateMachine.lfElapsed := Runtime(mem := "DB_Profiling".Section20_StateMachine.lfMemory);
   END_IF;
END_REGION

REGION Network 3: Alarms
   // no SCL statement known for Runtime: written as a call
   IF "DB_System".bProfiling THEN
       "DB_Profiling".Section20_ControlAlarmHandling.lfElapsed := Runtime(mem := "DB_Profiling".Section20_ControlAlarmHandling.lfMemory);
   END_IF;
   "ControlAlarmHandling_DB"();   // "ControlAlarmHandling"
   IF "DB_System".bProfiling THEN
       "DB_Profiling".Section20_ControlAlarmHandling.lfElapsed := Runtime(mem := "DB_Profiling".Section20_ControlAlarmHandling.lfMemory);
   END_IF;
END_REGION

REGION Network 4: Regulation
   // no SCL statement known for Runtime: written as a call
   IF "DB_System".bProfiling THEN
       "DB_Profiling".Section20_Regulation.lfElapsed := Runtime(mem := "DB_Profiling".Section20_Regulation.lfMemory);
   END_IF;
   "Regulation_DB"();   // "Regulation"
   IF "DB_System".bProfiling THEN
       "DB_Profiling".Section20_Regulation.lfElapsed := Runtime(mem := "DB_Profiling".Section20_Regulation.lfMemory);
   END_IF;
END_REGION

REGION Network 5: Start and stop
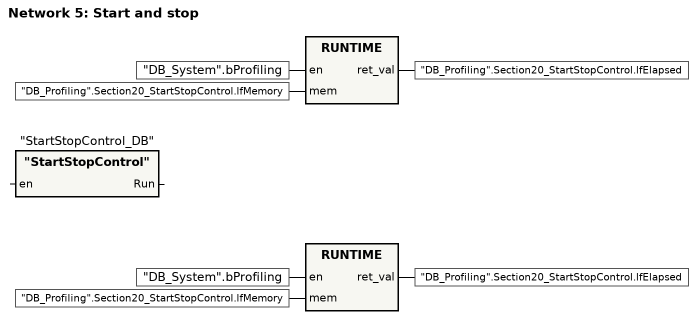
   // no SCL statement known for Runtime: written as a call
   IF "DB_System".bProfiling THEN
       "DB_Profiling".Section20_StartStopControl.lfElapsed := Runtime(mem := "DB_Profiling".Section20_StartStopControl.lfMemory);
   END_IF;
   "StartStopControl_DB"();   // "StartStopControl"
   IF "DB_System".bProfiling THEN
       "DB_Profiling".Section20_StartStopControl.lfElapsed := Runtime(mem := "DB_Profiling".Section20_StartStopControl.lfMemory);
   END_IF;
END_REGION
END_FUNCTION

FUNCTION_BLOCK "Calculations"   // FB42, FBD
{ S7_Optimized_Access := 'TRUE' }
VERSION : 0.1
// stored: AutoNumber true, IsIECCheckEnabled false, IsRetainMemResEnabled false, MemoryReserve 0, SetENOAutomatically false, UDAEnableTagReadback false
   VAR
      OperatingTimeCounters_Instance { ExternalAccessible := 'False'; ExternalVisible := 'False'; ExternalWritable := 'False'; S7_SetPoint := 'True'} : "OperatingTimeCounters";
      DT1_Merker_intern { ExternalAccessible := 'False'; ExternalVisible := 'False'; ExternalWritable := 'False'; S7_SetPoint := 'True'} : Real;
   END_VAR
   VAR_TEMP
      HeatRateSource : Real;
      HeatRateSink : Real;
      COP_max : Real;
      Quality : Real;
      COP : Real;
      HeatSourceDegreesPerSec : Real;
      HeatSourceDegreesPerMin : Real;
   END_VAR
   VAR_TEMP   // added for the SCL form of the ladder/FBD networks
      _w1 : Bool;
   END_VAR
BEGIN

REGION Network 1: Compressor calculations
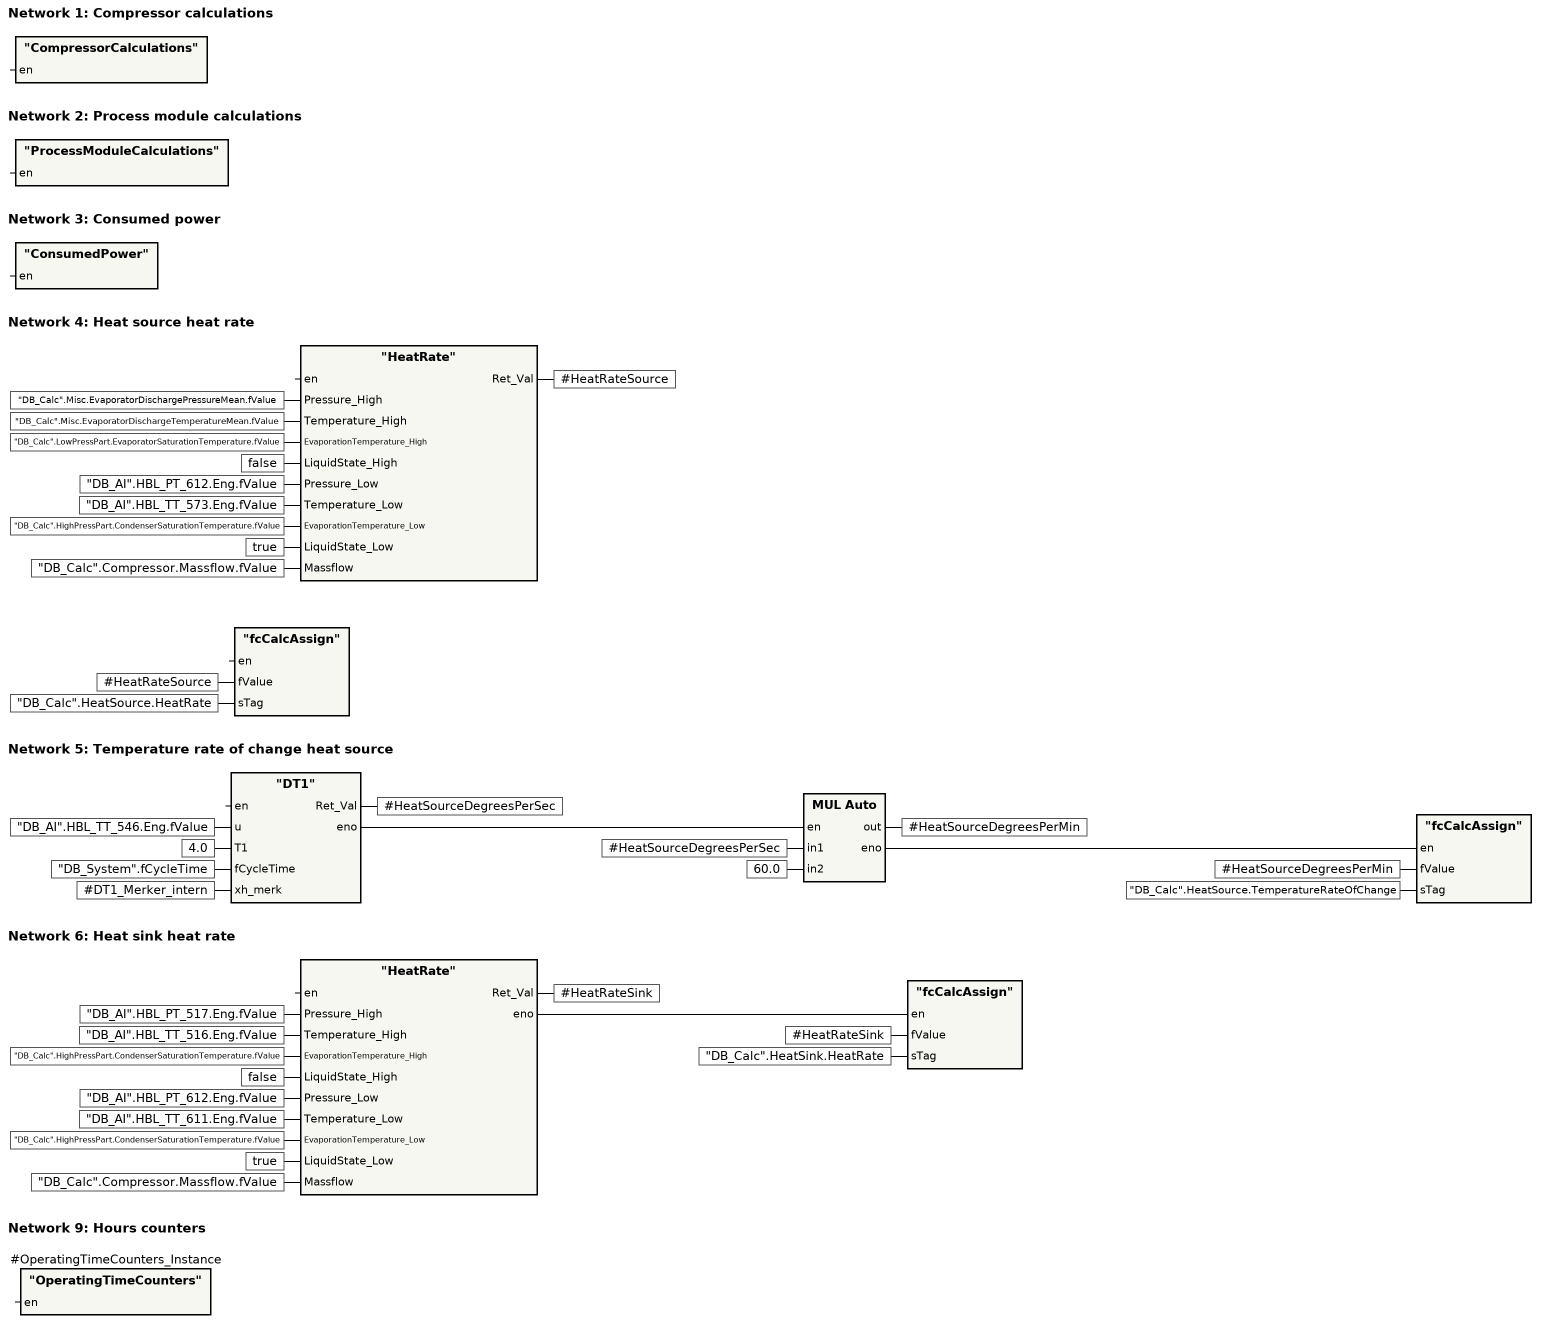
   "CompressorCalculations"();
END_REGION

REGION Network 2: Process module calculations
   "ProcessModuleCalculations"();
END_REGION

REGION Network 3: Consumed power
   "ConsumedPower"();
END_REGION

REGION Network 4: Heat source heat rate
   // The high side is the evaporator discharge temp & pressure, in gas phase
   // The low side, should be the evaporator suction temp & pressure, in liquid phase, but:
   //  - the condenser discharge pressure is used as it is the only pressure reading in that part of the system.
   //  - the expansion valve temperature is used
   // "We use the entalpy of the liquid before the expansion valve instead of the one before the evaporator, because the pressure and quality of the fluid before the evaporator is uncertain,  but it is known before the expansion valve and the expansion valve itself does not alter the enthalpy very much. "
   #HeatRateSource := "HeatRate"(Pressure_High := "DB_Calc".Misc.EvaporatorDischargePressureMean.fValue,
                           Temperature_High := "DB_Calc".Misc.EvaporatorDischargeTemperatureMean.fValue,
                           EvaporationTemperature_High := "DB_Calc".LowPressPart.EvaporatorSaturationTemperature.fValue,
                           LiquidState_High := false,
                           Pressure_Low := "DB_AI".HBL_PT_612.Eng.fValue,
                           Temperature_Low := "DB_AI".HBL_TT_573.Eng.fValue,
                           EvaporationTemperature_Low := "DB_Calc".HighPressPart.CondenserSaturationTemperature.fValue,
                           LiquidState_Low := true,
                           Massflow := "DB_Calc".Compressor.Massflow.fValue);
   "fcCalcAssign"(fValue := #HeatRateSource, sTag := "DB_Calc".HeatSource.HeatRate);
END_REGION

REGION Network 5: Temperature rate of change heat source
   // ###BE AWARE changed from K/sec to K/min
   #HeatSourceDegreesPerSec := "DT1"(u := "DB_AI".HBL_TT_546.Eng.fValue,
                           T1 := 4.0,
                           fCycleTime := "DB_System".fCycleTime,
                           xh_merk := #DT1_Merker_intern,
                           ENO => #_w1);
   IF #_w1 THEN
       #HeatSourceDegreesPerMin := #HeatSourceDegreesPerSec * 60.0;
       "fcCalcAssign"(fValue := #HeatSourceDegreesPerMin, sTag := "DB_Calc".HeatSource.TemperatureRateOfChange);
   END_IF;
END_REGION

REGION Network 6: Heat sink heat rate
   // The high side is the condenser suction temp & pressure, in gas phase
   // The low side is the condenser discharge temp & pressure, in liquid phase
   #HeatRateSink := "HeatRate"(Pressure_High := "DB_AI".HBL_PT_517.Eng.fValue,
                           Temperature_High := "DB_AI".HBL_TT_516.Eng.fValue,
                           EvaporationTemperature_High := "DB_Calc".HighPressPart.CondenserSaturationTemperature.fValue,
                           LiquidState_High := false,
                           Pressure_Low := "DB_AI".HBL_PT_612.Eng.fValue,
                           Temperature_Low := "DB_AI".HBL_TT_611.Eng.fValue,
                           EvaporationTemperature_Low := "DB_Calc".HighPressPart.CondenserSaturationTemperature.fValue,
                           LiquidState_Low := true,
                           Massflow := "DB_Calc".Compressor.Massflow.fValue,
                           ENO => #_w1);
   IF #_w1 THEN "fcCalcAssign"(fValue := #HeatRateSink, sTag := "DB_Calc".HeatSink.HeatRate); END_IF;
END_REGION

REGION Network 7 (SCL): COP
    IF "DB_Calc".System.ElectricalPower.fValue > 0.0 THEN
       #COP := "DB_Calc".HeatSink.HeatRate.fValue / "DB_Calc".System.ElectricalPower.fValue;
   ELSE
       #COP := 0.0;
   END_IF;

   "fcCalcAssign"(fValue := #COP, sTag := "DB_Calc".System.COP);
END_REGION

REGION Network 8 (SCL): Carnot quality
   // Quality rating is COP divided by COP_max (Carnot)
   // Verify this expression
   #COP_max := (("DB_AI".HBL_TT_901.Eng.fValue + "DB_AI".HBL_TT_518.Eng.fValue/2+273.15) * 
                ("DB_AI".HBL_TT_901.Eng.fValue + "DB_AI".HBL_TT_518.Eng.fValue -
                 "DB_AI".HBL_TT_542.Eng.fValue - "DB_AI".HBL_TT_546.Eng.fValue)/2 *100.0);

   IF "DB_AI".HBL_TT_542.Eng.fValue < "DB_AI".HBL_TT_901.Eng.fValue THEN
       #Quality := #COP / #COP_max;
   ELSE
       #Quality := 0.0;
   END_IF;

   "fcCalcAssign"(fValue := #Quality, sTag := "DB_Calc".System.Quality);
END_REGION

REGION Network 9: Hours counters
   #OperatingTimeCounters_Instance();   // "OperatingTimeCounters"
END_REGION

REGION Network 10: Temperature Lift
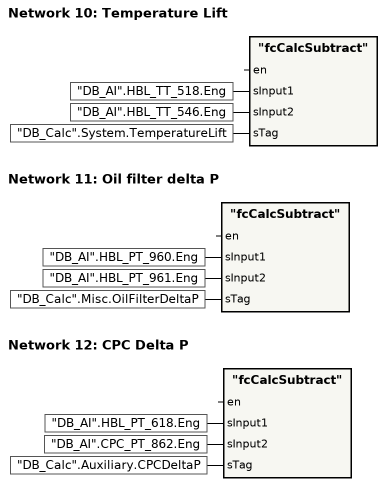
   "fcCalcSubtract"(sInput1 := "DB_AI".HBL_TT_518.Eng,
                    sInput2 := "DB_AI".HBL_TT_546.Eng,
                    sTag := "DB_Calc".System.TemperatureLift);
END_REGION

REGION Network 11: Oil filter delta P
   "fcCalcSubtract"(sInput1 := "DB_AI".HBL_PT_960.Eng,
                    sInput2 := "DB_AI".HBL_PT_961.Eng,
                    sTag := "DB_Calc".Misc.OilFilterDeltaP);
END_REGION

REGION Network 12: CPC Delta P
   // Actually the delta P over "orifice" V-861
   "fcCalcSubtract"(sInput1 := "DB_AI".HBL_PT_618.Eng,
                    sInput2 := "DB_AI".CPC_PT_862.Eng,
                    sTag := "DB_Calc".Auxiliary.CPCDeltaP);
END_REGION
END_FUNCTION_BLOCK

FUNCTION "CompressorCalculations" : Void   // FC25, FBD
{ S7_Optimized_Access := 'TRUE' }
VERSION : 0.1
// stored: AutoNumber true, IsIECCheckEnabled false, SetENOAutomatically false, UDAEnableTagReadback false
   VAR_TEMP
      CrankcaseSaturationTemperature : Real;
      SaturationTemperatureSuction : Real;
      SaturationTemperatureDischarge : Real;
      Massflow : Real;
      VolumetricEfficiency : Real;
      HeatRateCompressor : Real;
      IsentropicEfficiencyCompressor : Real;
      FMEP : Real;
   END_VAR
   VAR_TEMP   // added for the SCL form of the ladder/FBD networks
      _w1 : Bool;
   END_VAR
BEGIN

REGION Network 1: Crankcase saturation temperature
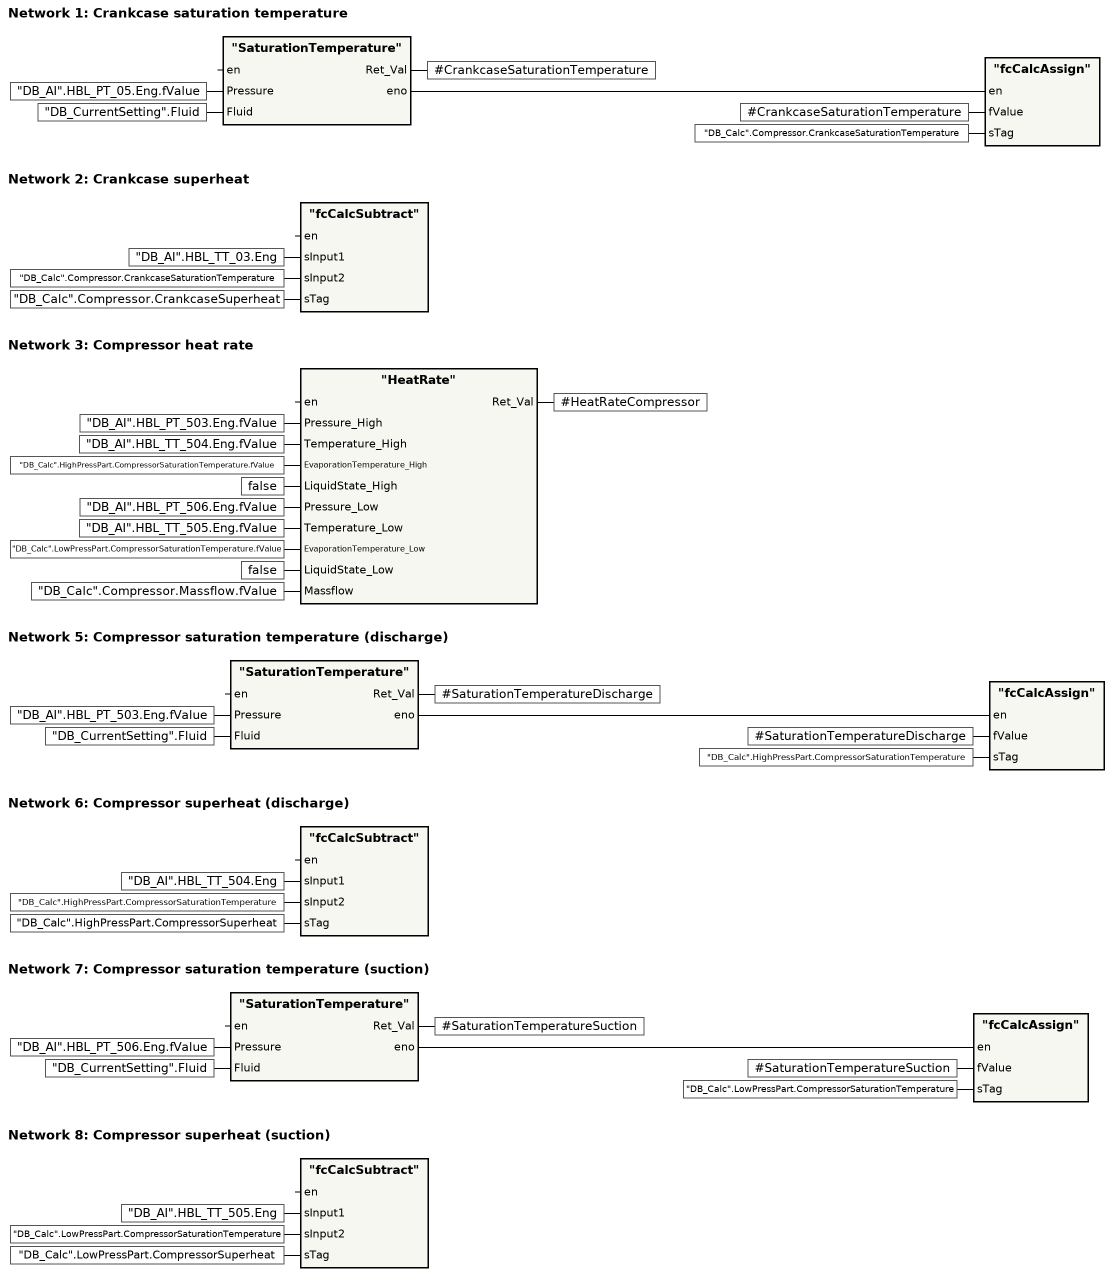
   #CrankcaseSaturationTemperature := "SaturationTemperature"(Pressure := "DB_AI".HBL_PT_05.Eng.fValue,
                           Fluid := "DB_CurrentSetting".Fluid,
                           ENO => #_w1);
   IF #_w1 THEN
       "fcCalcAssign"(fValue := #CrankcaseSaturationTemperature,
                      sTag := "DB_Calc".Compressor.CrankcaseSaturationTemperature);
   END_IF;
END_REGION

REGION Network 2: Crankcase superheat
   // Crankcase temperature is taken to be the same as the oil sump oil temperature
   "fcCalcSubtract"(sInput1 := "DB_AI".HBL_TT_03.Eng,
                    sInput2 := "DB_Calc".Compressor.CrankcaseSaturationTemperature,
                    sTag := "DB_Calc".Compressor.CrankcaseSuperheat);
END_REGION

REGION Network 3: Compressor heat rate
   // The high side is the compressor discharge temp & pressure, gas phase
   // The low side is the compressor suction temp & pressure, gas phase
   #HeatRateCompressor := "HeatRate"(Pressure_High := "DB_AI".HBL_PT_503.Eng.fValue,
                           Temperature_High := "DB_AI".HBL_TT_504.Eng.fValue,
                           EvaporationTemperature_High := "DB_Calc".HighPressPart.CompressorSaturationTemperature.fValue,
                           LiquidState_High := false,
                           Pressure_Low := "DB_AI".HBL_PT_506.Eng.fValue,
                           Temperature_Low := "DB_AI".HBL_TT_505.Eng.fValue,
                           EvaporationTemperature_Low := "DB_Calc".LowPressPart.CompressorSaturationTemperature.fValue,
                           LiquidState_Low := false,
                           Massflow := "DB_Calc".Compressor.Massflow.fValue);
END_REGION

REGION Network 4 (SCL): Isentropic efficiency
   IF "DB_Calc".System.ElectricalPower.fValue > 0.0 THEN
       #IsentropicEfficiencyCompressor := #HeatRateCompressor / "DB_Calc".System.ElectricalPower.fValue * 100.0;
   ELSE
       #IsentropicEfficiencyCompressor := 0.0;
   END_IF;

   "fcCalcAssign"(fValue := #IsentropicEfficiencyCompressor, sTag := "DB_Calc".Compressor.IsentropicEfficiency);
END_REGION

REGION Network 5: Compressor saturation temperature (discharge)
   // High press part
   #SaturationTemperatureDischarge := "SaturationTemperature"(Pressure := "DB_AI".HBL_PT_503.Eng.fValue,
                           Fluid := "DB_CurrentSetting".Fluid,
                           ENO => #_w1);
   IF #_w1 THEN
       "fcCalcAssign"(fValue := #SaturationTemperatureDischarge,
                      sTag := "DB_Calc".HighPressPart.CompressorSaturationTemperature);
   END_IF;
END_REGION

REGION Network 6: Compressor superheat (discharge)
   // Superheat out = Compressor discharge temperature - compressor saturation temperature
   "fcCalcSubtract"(sInput1 := "DB_AI".HBL_TT_504.Eng,
                    sInput2 := "DB_Calc".HighPressPart.CompressorSaturationTemperature,
                    sTag := "DB_Calc".HighPressPart.CompressorSuperheat);
END_REGION

REGION Network 7: Compressor saturation temperature (suction)
   #SaturationTemperatureSuction := "SaturationTemperature"(Pressure := "DB_AI".HBL_PT_506.Eng.fValue,
                           Fluid := "DB_CurrentSetting".Fluid,
                           ENO => #_w1);
   IF #_w1 THEN
       "fcCalcAssign"(fValue := #SaturationTemperatureSuction,
                      sTag := "DB_Calc".LowPressPart.CompressorSaturationTemperature);
   END_IF;
END_REGION

REGION Network 8: Compressor superheat (suction)
   // Superheat in = Compressor suction temperature - compressor saturation temperature
   "fcCalcSubtract"(sInput1 := "DB_AI".HBL_TT_505.Eng,
                    sInput2 := "DB_Calc".LowPressPart.CompressorSaturationTemperature,
                    sTag := "DB_Calc".LowPressPart.CompressorSuperheat);
END_REGION

REGION Network 9: Massflow & volumetric efficiency
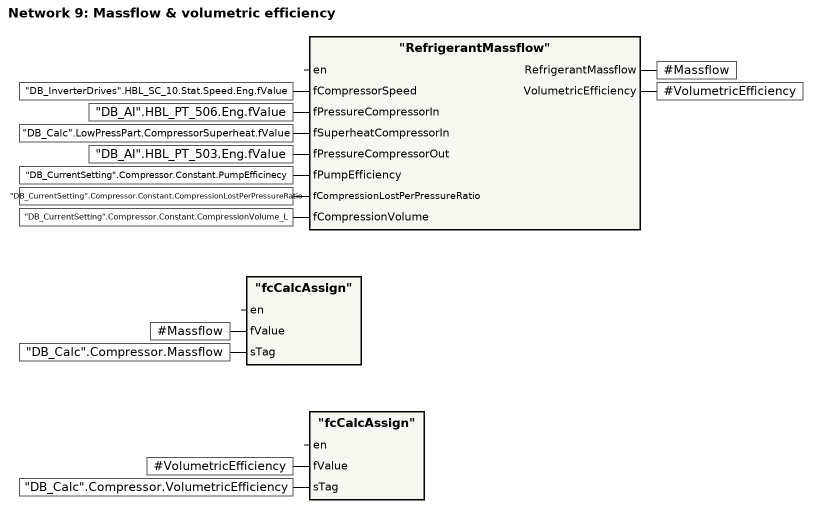
   "RefrigerantMassflow"(fCompressorSpeed := "DB_InverterDrives".HBL_SC_10.Stat.Speed.Eng.fValue,
                         fPressureCompressorIn := "DB_AI".HBL_PT_506.Eng.fValue,
                         fSuperheatCompressorIn := "DB_Calc".LowPressPart.CompressorSuperheat.fValue,
                         fPressureCompressorOut := "DB_AI".HBL_PT_503.Eng.fValue,
                         fPumpEfficiency := "DB_CurrentSetting".Compressor.Constant.PumpEfficinecy,
                         fCompressionLostPerPressureRatio := "DB_CurrentSetting".Compressor.Constant.CompressionLostPerPressureRatio,
                         fCompressionVolume := "DB_CurrentSetting".Compressor.Constant.CompressionVolume_L,
                         RefrigerantMassflow => #Massflow,
                         VolumetricEfficiency => #VolumetricEfficiency);
   "fcCalcAssign"(fValue := #Massflow, sTag := "DB_Calc".Compressor.Massflow);
   "fcCalcAssign"(fValue := #VolumetricEfficiency, sTag := "DB_Calc".Compressor.VolumetricEfficiency);
END_REGION

REGION Network 10 (SCL): FMEP
   // IMEP is estimated as follows:
   // IMEP ~(discharge pressure + suction pressure)/2
   // BMEP = Torque * 0.37793 kPa/Nm
   // FMEP = IMEP - BMEP
   // FMEP = (discharge pressure + suction pressure)/2 - Torque * 0.37793 kPa/Nm

   #FMEP := ("DB_AI".HBL_PT_506.Eng.fValue + "DB_AI".HBL_PT_503.Eng.fValue)/2 - "DB_InverterDrives".HBL_SC_10.Stat.Torque.Eng.fValue/100 * 3407 * 0.37793;
   "fcCalcAssign"(fValue := #FMEP, sTag := "DB_Calc".System.FMEP);
END_REGION
END_FUNCTION

FUNCTION "SaturationTemperature" : Real   // FC14, FBD
{ S7_Optimized_Access := 'TRUE' }
VERSION : 0.1
// stored: AutoNumber true, IsIECCheckEnabled false, SetENOAutomatically false, UDAEnableTagReadback false
   VAR_INPUT
      Pressure : Real;
   END_VAR
   VAR_IN_OUT
      Fluid : "FluidData-STRUCT";
   END_VAR
   VAR_TEMP
      MinPressure : Real;
   END_VAR
BEGIN

REGION Network 1
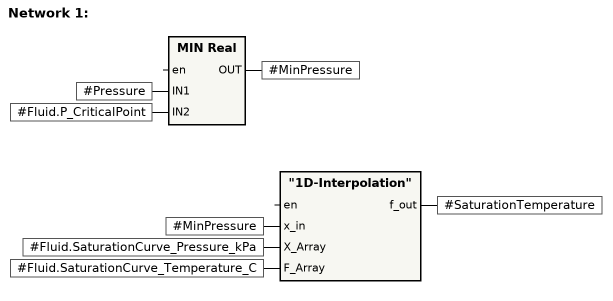
   #MinPressure := MIN(IN1 := #Pressure, IN2 := #Fluid.P_CriticalPoint);
   "1D-Interpolation"(x_in := #MinPressure,
                      X_Array := #Fluid.SaturationCurve_Pressure_kPa,
                      F_Array := #Fluid.SaturationCurve_Temperature_C,
                      f_out => #SaturationTemperature);
END_REGION
END_FUNCTION

FUNCTION "1D-Interpolation" : Void
{ S7_Optimized_Access := 'TRUE' }
VERSION : 0.1
   VAR_INPUT 
      x_in : Real;
   END_VAR

   VAR_OUTPUT 
      f_out : Real;
   END_VAR

   VAR_IN_OUT 
      X_Array : Array[*] of Real;
      F_Array : Array[*] of Real;
   END_VAR

   VAR_TEMP 
      Xindex_L : DInt;
      X_L : Real;
      X_H : Real;
      F_Lx : Real;
      F_Hx : Real;
      x : Real;
   END_VAR


BEGIN
	#x := #x_in;
	
	"FindIndex"(x:=#x,
	            index_L=>#Xindex_L,
	            Array:=#X_Array);
	(* REGION Find nearest meshpoint (#X_Array[#index_Lx]) smaller than x
	    // If x is closest to the last index or lies beyond, then take the second last index anyway
	    // We use our previous result from last calculation (#LastIndexNr) as startpoint for the search
	    #Xindex_L := #LastXi;
	    IF #Xindex_L > 0 AND #x < #X_Array[#Xindex_L] THEN
	        //Suche nach links (kleinere indizes)
	        WHILE #Xindex_L > 0 AND #x < #X_Array[#Xindex_L - 1] DO
	            #Xindex_L -= 1;
	            IF #Xindex_L = 0 THEN
	                EXIT;
	            END_IF;
	        END_WHILE;
	    ELSE
	        //Suche nach rechts (größere indizes)
	        WHILE #Xindex_L < (#Count_Xi - 1) AND #x > #X_Array[#Xindex_L + 1] DO
	            #Xindex_L += 1;
	        END_WHILE;
	    END_IF;
	END_REGION *)
	
	
	REGION interpolation points    
	    // The interpolation points are:
	    #X_L := #X_Array[#Xindex_L];   //The largest meshpoint smaller larger than x (< Count_X-1)
	    #X_H := #X_Array[#Xindex_L + 1]; //The smalles meshpoint bigger larger than x  (>= 1)
	    #F_Lx := #F_Array[#Xindex_L];  // Function value of X_L
	    #F_Hx := #F_Array[#Xindex_L + 1];// Function value of X_H
	    IF #X_L >= #X_H THEN // The lookup has rise strictly monotonously
	        ENO := 1;
	        #f_out := "NaN"();
	        RETURN;
	    END_IF;
	END_REGION
	
	REGION inerpolation
	    //Calculate interpolation inbetween or beyond X_L and X_H
	    #f_out := (#F_Hx - #F_Lx) / (#X_H - #X_L) * (#x - #X_L) + #F_Lx;
	END_REGION
	
END_FUNCTION

FUNCTION "FindIndex" : Void
{ S7_Optimized_Access := 'TRUE' }
VERSION : 0.1
   VAR_INPUT 
      x : Real;
   END_VAR

   VAR_OUTPUT 
      index_L : DInt;
   END_VAR

   VAR_IN_OUT 
      "Array" : Array[*] of Real;
   END_VAR

   VAR_TEMP 
      Count_i : DInt;
   END_VAR


BEGIN
	        
	        
	        #Count_i := UPPER_BOUND(ARR:=#Array, DIM:=1);
	        #index_L := #Count_i/2;
	    // If x is closest to the last index (Count_Xi) or lies beyond, then take the second last index anyway
	    // We use our previous result from last calculation (#LastXi) as startpoint for the search
	    //#Xindex_L := #LastXi;
	    //IF #index_L > 0 AND #x < #Array[#index_L] THEN //die If ist nicht unbedingt notwendig.
	        //Suche nach links (kleinere indizes)
	        WHILE #index_L > 0 AND #x < #Array[#index_L] DO
	            #index_L -= 1;
	            //IF #index_L = 0 THEN // Durch Schleifenbedingung unnötig, oder?!
	            //    EXIT;
	            //END_IF;
	        END_WHILE;
	    //ELSE
	    //Suche nach rechts (größere indizes)
	        WHILE #index_L < (#Count_i - 1) AND #x > #Array[#index_L + 1] DO
	            #index_L += 1;
	        END_WHILE;
	    //END_IF;
END_FUNCTION

FUNCTION "HeatRate" : Real
{ S7_Optimized_Access := 'TRUE' }
VERSION : 0.1
   VAR_INPUT 
      Pressure_High : Real;   // Bar
      Temperature_High : Real;   // C
      EvaporationTemperature_High : Real;   // C
      LiquidState_High : Bool;   // 1 = liquid, 0 = gas
      Pressure_Low : Real;   // Bar
      Temperature_Low : Real;   // C
      EvaporationTemperature_Low : Real;   // C
      LiquidState_Low : Bool;   // 1 = liquid, 0 = gas
      Massflow : Real;   // kg/h
   END_VAR

   VAR_TEMP 
      H_High : Real;   // High value of Enthalpy
      H_Low : Real;   // Low value of Enthalpy
   END_VAR


BEGIN
	// The difference of the enthalpy values times massflow is the heat rate Qdot
	// Use the "High" group of values for the side of the enthalpy source/sink with the greatest magnitude, so as to get positive values
	
	#H_High := "Enthalpy_f"(Pressure := #Pressure_High,
	                        Themperature := #Temperature_High,
	                        EvaporationTemperature := #EvaporationTemperature_High, 
	                        Gas := NOT #LiquidState_High, 
	                        Liquide := #LiquidState_High);
	    
	#H_Low := "Enthalpy_f"(Pressure := #Pressure_Low,  
	                       Themperature := #Temperature_Low,
	                       EvaporationTemperature := #EvaporationTemperature_Low, 
	                       Gas := NOT #LiquidState_Low, 
	                       Liquide := #LiquidState_Low);
	
	// Convert Massflow into kg/s
	#HeatRate := (#H_High - #H_Low) * (#Massflow / 3600.0);
END_FUNCTION

FUNCTION "Enthalpy_f" : Real
{ S7_Optimized_Access := 'TRUE' }
VERSION : 0.1
   VAR_INPUT 
      Pressure : Real;
      Themperature : Real;
      EvaporationTemperature : Real;
      Gas : Bool;
      Liquide : Bool;
   END_VAR

   VAR_TEMP 
      Superheat : Real;
   END_VAR

   VAR CONSTANT 
      Lim : Real := 0.01;
   END_VAR


BEGIN
	#Superheat := #Themperature-#EvaporationTemperature;
	IF #Gas THEN
	    #Superheat := MAX(IN1:=#Superheat, IN2:=#Lim);
	ELSIF #Liquide THEN
	    #Superheat := MIN(IN1:=#Superheat, IN2:=-#Lim);
	END_IF;
	
	"2D-Interpolation"(x_in:=#Pressure,
	                         y_in:=#Superheat,
	                         f_out=>#Enthalpy_f,
	                         X_Array:="DB_CurrentSetting".Fluid.EnthalpyMap_Pressure_kPa,
	                         Y_Array:="DB_CurrentSetting".Fluid.EnthalpyMap_Superheat_C,
	                         F_Array:="DB_CurrentSetting".Fluid.EnthalpyMap_Enthalpy_kJ_kg);
	ENO := ENO;
END_FUNCTION

FUNCTION "2D-Interpolation" : Void
{ S7_Optimized_Access := 'TRUE' }
VERSION : 0.1
   VAR_INPUT 
      x_in : Real;
      y_in : Real;
   END_VAR

   VAR_OUTPUT 
      f_out : Real;
   END_VAR

   VAR_IN_OUT 
      X_Array : Array[*] of Real;
      Y_Array : Array[*] of Real;
      F_Array : Array[*, *] of Real;
   END_VAR

   VAR_TEMP 
      Xindex_L : DInt;
      Xindex_U : DInt;
      Yindex_L : DInt;
      Yindex_U : DInt;
      X_L : Real;
      X_H : Real;
      Y_L : Real;
      Y_H : Real;
      F_LxLy : Real;
      F_LxHy : Real;
      F_HxLy : Real;
      F_HxHy : Real;
      x : Real;
      y : Real;
   END_VAR


BEGIN
	#x := #x_in;
	#y := #y_in;
	
	"FindIndex"(x:=#x,
	            index_L=>#Xindex_L,
	            Array:=#X_Array);
	"FindIndex"(x:=#y,
	            index_L=>#Yindex_L,
	            Array:=#Y_Array);
	(* REGION Find nearest meshpoint (#Y_Array[#Xindex_L]) smaller than x
	    // If x is closest to the last index (Count_Xi) or lies beyond, then take the second last index anyway
	    // We use our previous result from last calculation (#LastXi) as startpoint for the search
	    #Xindex_L := #LastXi;
	    IF #Xindex_L > 0 AND #x < #X_Array[#Xindex_L] THEN
	        //Suche nach links (kleinere indizes)
	        WHILE #Xindex_L > 0 AND #x < #X_Array[#Xindex_L - 1] DO
	            #Xindex_L -= 1;
	            IF #Xindex_L = 0 THEN
	                EXIT;
	            END_IF;
	        END_WHILE;
	    ELSE
	        //Suche nach rechts (größere indizes)
	        WHILE #Xindex_L < (#Count_Xi - 1) AND #x > #X_Array[#Xindex_L + 1] DO
	            #Xindex_L += 1;
	        END_WHILE;
	    END_IF;
	END_REGION
	REGION Find nearest meshpoint (#Y_Array[#Yindex_L]) smaller than y
	    // If y is closest to the last index (count_Yi) or lies beyond, then take the second last index anyway
	    // We use our previous result from last calculation (#LastYi) as startpoint for the search
	    #Yindex_L := #LastYi;
	    IF #Yindex_L > 0 AND #y < #Y_Array[#Yindex_L] THEN
	        //Suche nach links (kleinere indizes)
	        WHILE #Yindex_L > 0 AND #y < #Y_Array[#Yindex_L - 1] DO
	            #Yindex_L -= 1;
	            IF #Yindex_L = 0 THEN
	                EXIT;
	            END_IF;
	        END_WHILE;
	    ELSE
	        //Suche nach rechts (größere indizes)
	        WHILE #Yindex_L < (#Count_Yi - 1) AND #y > #Y_Array[#Yindex_L + 1] DO
	            #Yindex_L += 1;
	        END_WHILE;
	    END_IF;
	END_REGION*) //Replaced by "Function"
	#Xindex_U := #Xindex_L +1;
	#Yindex_U := #Yindex_L +1;
	
	REGION interpolation points    
	    // The interpolation points are:
	
	    
	    #X_L := #X_Array[#Xindex_L]; //The largest meshpoint smaller larger than x (< Count_Xi-1)
	    #X_H := #X_Array[#Xindex_U]; //The smalles meshpoint bigger larger than x  (>= 1)
	    #Y_L := #Y_Array[#Yindex_L]; //The largest meshpoint smaller larger than x (< Count_Xi-1)
	    #Y_H := #Y_Array[#Yindex_U]; //The smalles meshpoint bigger larger than x  (>= 1)
	    #F_LxLy := #F_Array[#Xindex_L, #Yindex_L]; // Function value of (X_L,X_L)
	    #F_LxHy := #F_Array[#Xindex_L, #Yindex_U]; // Function value of (X_L,X_H)
	    #F_HxLy := #F_Array[#Xindex_U, #Yindex_L]; // Function value of (X_L,X_L)
	    #F_HxHy := #F_Array[#Xindex_U, #Yindex_U]; // Function value of (X_L,X_H)
	    
	    IF #X_L >= #X_H AND #Y_L >= #Y_H THEN // The lookup has rise strictly monotonously
	        ENO := 1;
	        #f_out := "NaN"();
	        RETURN;
	    END_IF;
	END_REGION
	
	REGION inerpolation
	    //Calculate interpolation with the four meshpoints (X_L,Y_L) (X_H,Y_L) (X_L,Y_H) and (X_H,Y_H)
	    #x:= (#x - #X_L) / (#X_H - #X_L);
	    #y:= (#y - #Y_L) / (#Y_H - #Y_L);
	    #f_out := (#F_HxLy - #F_LxLy) * #x;
	    #f_out += (#F_HxHy - #F_HxLy) * #y;
	    #f_out += (#F_LxHy - #F_LxLy) * #y;
	    #f_out += (#F_HxHy - #F_LxHy) * #x;
	    #f_out /= 2.0;
	    #f_out += #F_LxLy;
	  (*  #f_out :=
	    (#F_HxLy - #F_LxLy) / (#X_H - #X_L) * (#x - #X_L) / 2 +
	    (#F_HxHy - #F_HxLy) / (#Y_H - #Y_L) * (#y - #Y_L) / 2 +
	    (#F_LxHy - #F_LxLy) / (#Y_H - #Y_L) * (#y - #Y_L) / 2 +
	    (#F_HxHy - #F_LxHy) / (#X_H - #X_L) * (#x - #X_L) / 2 +
	    #F_LxLy; *)
	    //There is still an unused information in there, witch can be used for an additional quadratic therm in the direction (X_L,Y_L)->(X_H,Y,H) or right-angled to it. 
	END_REGION
	
	
END_FUNCTION

FUNCTION "RefrigerantMassflow" : Void
{ S7_Optimized_Access := 'TRUE' }
VERSION : 0.1
   VAR_INPUT 
      fCompressorSpeed : Real;   // [rpm]
      fPressureCompressorIn : Real;   // [kPa]
      fSuperheatCompressorIn : Real;   // [C]
      fPressureCompressorOut : Real;   // [kPa]
      fPumpEfficiency : Real;   // [%]
      fCompressionLostPerPressureRatio : Real;   // [%]
      fCompressionVolume : Real;   // [L]
   END_VAR

   VAR_OUTPUT 
      RefrigerantMassflow : Real;   // [kg/h]
      VolumetricEfficiency : Real;   // [%]
   END_VAR

   VAR_TEMP 
      DensityCompressorIn : Real;   // [kg/m^3]
      VolEfficiency : Real;
      PressureRatio : Real;   // [1]
      "SystemVolumeFlow_m³/h" : Real;   // [m^3/h]
   END_VAR


BEGIN
	// Volumetric efficiency
	#PressureRatio := #fPressureCompressorOut / #fPressureCompressorIn;
	IF ENO = 0 THEN
	    #PressureRatio := 1.0;
	    ENO := 1;
	END_IF;
	
	#VolEfficiency := #fPumpEfficiency/100.0 - (#PressureRatio - 1.0) * #fCompressionLostPerPressureRatio/100.0;
	#VolumetricEfficiency := #VolEfficiency * 100.0;
	
	// Mass flow
	#"SystemVolumeFlow_m³/h" := #fCompressorSpeed * 60.0 * #fCompressionVolume * #VolEfficiency /1000.0;
	
	"DensityCompressorInlet"(fPressureCompressorIn:= #fPressureCompressorIn,
	                         fSuperheatCompresorIn:= #fSuperheatCompressorIn,
	                         fDensity=> #DensityCompressorIn);
	
	#RefrigerantMassflow := #"SystemVolumeFlow_m³/h" * #DensityCompressorIn;
	
END_FUNCTION

FUNCTION "DensityCompressorInlet" : Void
{ S7_Optimized_Access := 'TRUE' }
VERSION : 0.1
   VAR_INPUT 
      fPressureCompressorIn : Real;   // Bar
      fSuperheatCompresorIn : Real;   // C
   END_VAR

   VAR_OUTPUT 
      fDensity : Real;
   END_VAR


BEGIN
	"1D-Interpolation"(x_in:=#fPressureCompressorIn,
	                       f_out=>#fDensity,
	                       X_Array:="DB_CurrentSetting".Fluid.DensityCurve_Pressure_kPa,
	                       F_Array:="DB_CurrentSetting".Fluid.DensityCurveVapor_Densety_kg_m3);
	   
	   // Superheat Correction roh_corr = roh - (p²a+pb)*Tsuper
	   #fDensity -= (SQR(#fPressureCompressorIn) * "DB_CurrentSetting".Fluid.DensityCurveVapor_SuperheatCorrection_a + #fPressureCompressorIn * "DB_CurrentSetting".Fluid.DensityCurveVapor_SuperheatCorrection_b) * #fSuperheatCompresorIn;
END_FUNCTION

FUNCTION "ProcessModuleCalculations" : Void   // FC16, FBD
{ S7_Optimized_Access := 'TRUE' }
VERSION : 0.1
// stored: AutoNumber true, IsIECCheckEnabled false, SetENOAutomatically false, UDAEnableTagReadback false
   VAR_TEMP
      T_Evaporation_LP : Real;
      T_Condense_HP : Real;
   END_VAR
   VAR_TEMP   // added for the SCL form of the ladder/FBD networks
      _w1 : Bool;
   END_VAR
BEGIN

REGION Network 1: Evaporator discharge pressure mean
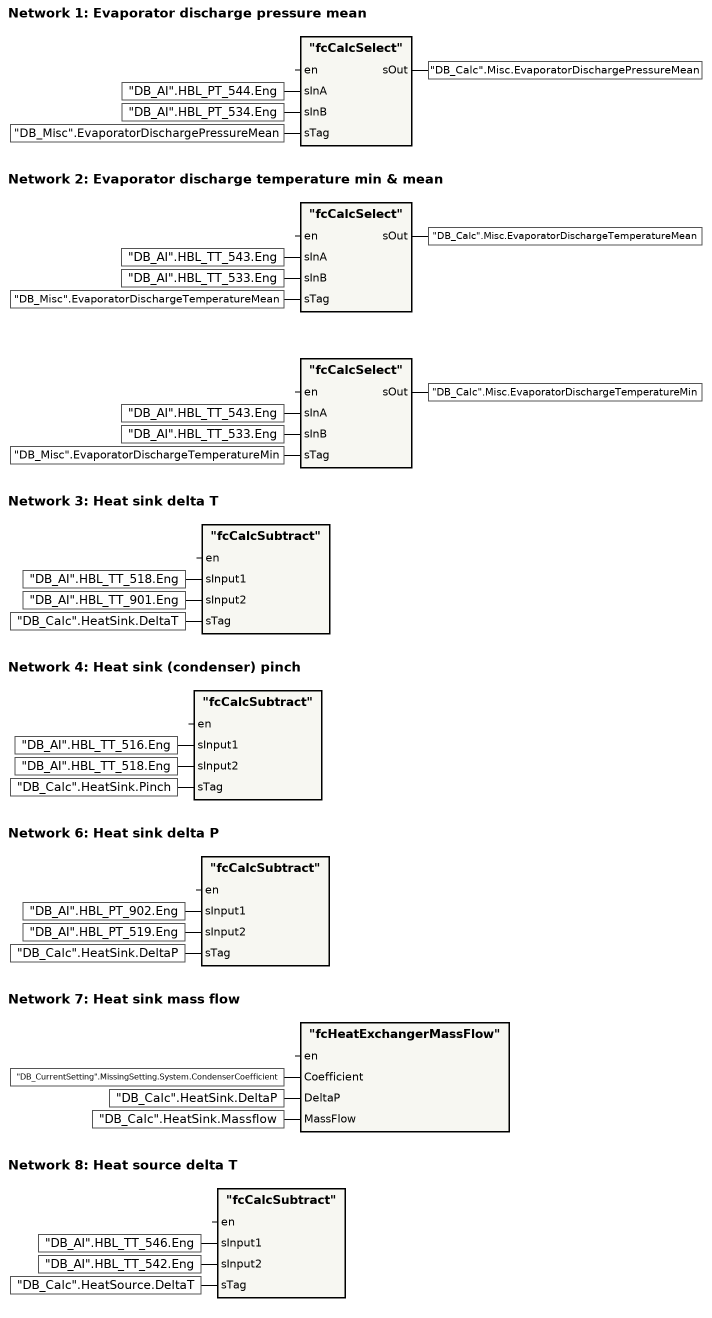
   "fcCalcSelect"(sInA := "DB_AI".HBL_PT_544.Eng,
                  sInB := "DB_AI".HBL_PT_534.Eng,
                  sTag := "DB_Misc".EvaporatorDischargePressureMean,
                  sOut => "DB_Calc".Misc.EvaporatorDischargePressureMean);
END_REGION

REGION Network 2: Evaporator discharge temperature min & mean
   "fcCalcSelect"(sInA := "DB_AI".HBL_TT_543.Eng,
                  sInB := "DB_AI".HBL_TT_533.Eng,
                  sTag := "DB_Misc".EvaporatorDischargeTemperatureMean,
                  sOut => "DB_Calc".Misc.EvaporatorDischargeTemperatureMean);
   "fcCalcSelect"(sInA := "DB_AI".HBL_TT_543.Eng,
                  sInB := "DB_AI".HBL_TT_533.Eng,
                  sTag := "DB_Misc".EvaporatorDischargeTemperatureMin,
                  sOut => "DB_Calc".Misc.EvaporatorDischargeTemperatureMin);
END_REGION

REGION Network 3: Heat sink delta T
   // Temperature rise (positive)
   "fcCalcSubtract"(sInput1 := "DB_AI".HBL_TT_518.Eng,
                    sInput2 := "DB_AI".HBL_TT_901.Eng,
                    sTag := "DB_Calc".HeatSink.DeltaT);
END_REGION

REGION Network 4: Heat sink (condenser) pinch
   // Pinch feed flow = Condenser suction temperature - Heat sink discharge temperature
   "fcCalcSubtract"(sInput1 := "DB_AI".HBL_TT_516.Eng,
                    sInput2 := "DB_AI".HBL_TT_518.Eng,
                    sTag := "DB_Calc".HeatSink.Pinch);
END_REGION

REGION Network 5: Heat sink heat rate
END_REGION

REGION Network 6: Heat sink delta P
   // Estimated from pressure drop across the condenser
   "fcCalcSubtract"(sInput1 := "DB_AI".HBL_PT_902.Eng,
                    sInput2 := "DB_AI".HBL_PT_519.Eng,
                    sTag := "DB_Calc".HeatSink.DeltaP);
END_REGION

REGION Network 7: Heat sink mass flow
   "fcHeatExchangerMassFlow"(Coefficient := "DB_CurrentSetting".MissingSetting.System.CondenserCoefficient,
                           DeltaP := "DB_Calc".HeatSink.DeltaP,
                           MassFlow := "DB_Calc".HeatSink.Massflow);
END_REGION

REGION Network 8: Heat source delta T
   // Temperature drop (positive)
   "fcCalcSubtract"(sInput1 := "DB_AI".HBL_TT_546.Eng,
                    sInput2 := "DB_AI".HBL_TT_542.Eng,
                    sTag := "DB_Calc".HeatSource.DeltaT);
END_REGION

REGION Network 9: Heat source pinch (evaporator)
   // Pinch return flow = Heat Source discharge temperature - Evaporation temperature
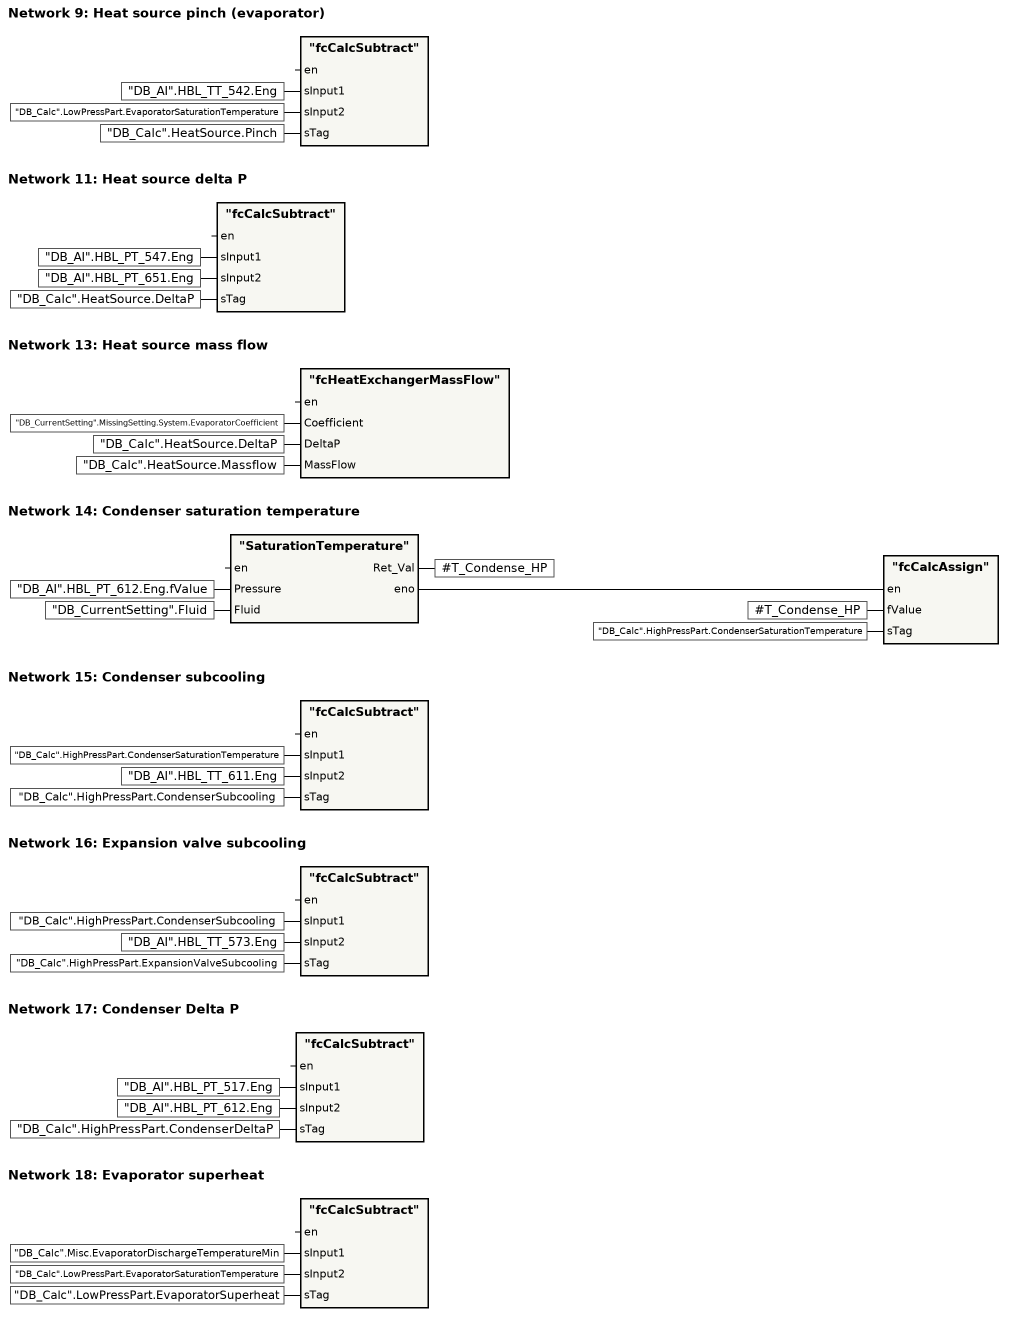
   "fcCalcSubtract"(sInput1 := "DB_AI".HBL_TT_542.Eng,
                    sInput2 := "DB_Calc".LowPressPart.EvaporatorSaturationTemperature,
                    sTag := "DB_Calc".HeatSource.Pinch);
END_REGION

REGION Network 10: Heat source heat rate
END_REGION

REGION Network 11: Heat source delta P
   // ##Note: this may not make a lot of sense. PT-547 is steam pressure, PT-651 is condensate pressure
   "fcCalcSubtract"(sInput1 := "DB_AI".HBL_PT_547.Eng,
                    sInput2 := "DB_AI".HBL_PT_651.Eng,
                    sTag := "DB_Calc".HeatSource.DeltaP);
END_REGION

REGION Network 12: Heat source temperature rate of change
   // in Calculations (FB42) as it requires static variables
END_REGION

REGION Network 13: Heat source mass flow
   "fcHeatExchangerMassFlow"(Coefficient := "DB_CurrentSetting".MissingSetting.System.EvaporatorCoefficient,
                           DeltaP := "DB_Calc".HeatSource.DeltaP,
                           MassFlow := "DB_Calc".HeatSource.Massflow);
END_REGION

REGION Network 14: Condenser saturation temperature
   #T_Condense_HP := "SaturationTemperature"(Pressure := "DB_AI".HBL_PT_612.Eng.fValue,
                           Fluid := "DB_CurrentSetting".Fluid,
                           ENO => #_w1);
   IF #_w1 THEN
       "fcCalcAssign"(fValue := #T_Condense_HP, sTag := "DB_Calc".HighPressPart.CondenserSaturationTemperature);
   END_IF;
END_REGION

REGION Network 15: Condenser subcooling
   "fcCalcSubtract"(sInput1 := "DB_Calc".HighPressPart.CondenserSaturationTemperature,
                    sInput2 := "DB_AI".HBL_TT_611.Eng,
                    sTag := "DB_Calc".HighPressPart.CondenserSubcooling);
END_REGION

REGION Network 16: Expansion valve subcooling
   "fcCalcSubtract"(sInput1 := "DB_Calc".HighPressPart.CondenserSubcooling,
                    sInput2 := "DB_AI".HBL_TT_573.Eng,
                    sTag := "DB_Calc".HighPressPart.ExpansionValveSubcooling);
END_REGION

REGION Network 17: Condenser Delta P
   "fcCalcSubtract"(sInput1 := "DB_AI".HBL_PT_517.Eng,
                    sInput2 := "DB_AI".HBL_PT_612.Eng,
                    sTag := "DB_Calc".HighPressPart.CondenserDeltaP);
END_REGION

REGION Network 18: Evaporator superheat
   "fcCalcSubtract"(sInput1 := "DB_Calc".Misc.EvaporatorDischargeTemperatureMin,
                    sInput2 := "DB_Calc".LowPressPart.EvaporatorSaturationTemperature,
                    sTag := "DB_Calc".LowPressPart.EvaporatorSuperheat);
END_REGION

REGION Network 19: Evaporator saturation temperature
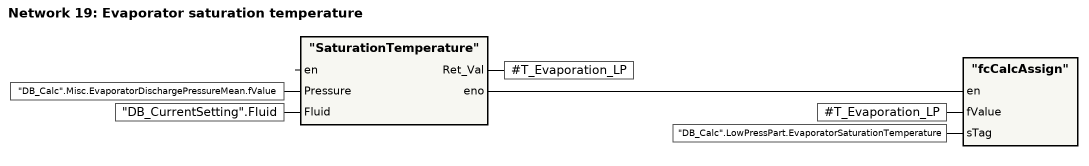
   #T_Evaporation_LP := "SaturationTemperature"(Pressure := "DB_Calc".Misc.EvaporatorDischargePressureMean.fValue,
                           Fluid := "DB_CurrentSetting".Fluid,
                           ENO => #_w1);
   IF #_w1 THEN
       "fcCalcAssign"(fValue := #T_Evaporation_LP, sTag := "DB_Calc".LowPressPart.EvaporatorSaturationTemperature);
   END_IF;
END_REGION
END_FUNCTION

FUNCTION "fcCalcSelect" : Void
{ S7_Optimized_Access := 'TRUE' }
VERSION : 0.1
   VAR_INPUT 
      sInA : "stCalcValue";   // First value
      sInB : "stCalcValue";   // Second value
   END_VAR

   VAR_OUTPUT 
      sOut : "stCalcValue";   // Result value
   END_VAR

   VAR_IN_OUT 
      sTag : "stCalcSelect";
   END_VAR

   VAR_TEMP 
      Avg : Real;
   END_VAR


BEGIN
	// fcCalcSelect - process two Calc values according to Mode.
	// Falls back to "best effort" if one of the inputs has .bError set
	
	// Modes: 
	// 0: none selected (off)
	// 1: Select A
	// 2: Select B
	// 3: MIN value
	// 4: MAX value
	// 5: Average value
	// 128: Error
	
	// Preprocessing in case of value error
	IF #sInA.bError = TRUE AND #sInB.bError = TRUE THEN
	    #sTag.nActualMode := 128;
	    #sTag.bError := TRUE;
	ELSIF #sInA.bError = FALSE AND #sInB.bError = TRUE THEN
	    #sTag.nActualMode := 1;
	    #sTag.bError := FALSE;
	ELSIF #sInA.bError = TRUE AND #sInB.bError = FALSE THEN
	    #sTag.nActualMode := 2;
	    #sTag.bError := FALSE;
	ELSE    
	    #sTag.nActualMode := #sTag.nMode;
	    #sTag.bError := FALSE;
	END_IF;
	
	// Choose value
	CASE #sTag.nActualMode OF
	    0: // neither selected, output a null value
	        #sOut.fMin := 0;
	        #sOut.fMax := 0;
	        "fcCalcAssign"(fValue := 0, sTag := #sOut);
	    1: // Select A
	        #sOut := #sInA;
	    2: // Select B
	        #sOut := #sInB;
	    3: // Select MIN
	        IF #sInA.fValue <= #sInB.fValue THEN
	            #sOut := #sInA;
	        ELSE
	            #sOut := #sInB;
	        END_IF;
	    4: // Select MAX
	        IF #sInA.fValue >= #sInB.fValue THEN
	            #sOut := #sInA;
	        ELSE
	            #sOut := #sInB;
	        END_IF;
	    5: // Select AVG
	         #Avg := (#sInA.fValue + #sInB.fValue)/2;
	        "fcCalcAssign"(fValue := #Avg, sTag := #sOut);
	    ELSE
	        // both in error
	        "fcCalcAssign"(fValue := "NaN"(), sTag := #sOut);
	END_CASE;
	
	// Warning
	#sTag.bWarning := (#sTag.nMode <> #sTag.nActualMode);
	
END_FUNCTION

FUNCTION "fcHeatExchangerMassFlow" : Void
{ S7_Optimized_Access := 'TRUE' }
VERSION : 0.1
   VAR_INPUT 
      Coefficient : Real;   // kPa to T/h conversion factor
      DeltaP : "stCalcValue";   // kPa
   END_VAR

   VAR_IN_OUT 
      MassFlow : "stCalcValue";
   END_VAR


BEGIN
	// Calculate mass flow through a heat exchanger from pressure drop
	
	IF #DeltaP.bError = TRUE THEN
	    "fcCalcAssign"(fValue := "NaN"(), sTag := #MassFlow);
	ELSE
	    "fcCalcAssign"(fValue := #Coefficient * SQRT(#DeltaP.fValue), sTag := #MassFlow);
	END_IF;
	
END_FUNCTION

FUNCTION "ConsumedPower" : Void   // FC20, FBD
TITLE = Tally up consumers
{ S7_Optimized_Access := 'TRUE' }
VERSION : 0.1
// stored: AutoNumber true, IsIECCheckEnabled false, SetENOAutomatically false, UDAEnableTagReadback false
   VAR_TEMP
      fPower : Real;
   END_VAR
   VAR CONSTANT
      SSC_P_01_POWER : Real := 0.55;   // kW
      SSC_P_02_POWER : Real := 0.55;   // kW
      SSC_F_01_POWER : Real := 0.55;   // kW
      CPC_P_01_POWER : Real := 1.1;   // kW
      CabinetHeater_POWER : Real := 0.045;   // kW
      CabinetFan_POWER : Real := 0.1;   // kW
      HBL_EC_01_POWER : Real := 4.0;   // kW
      HBL_EC_02_POWER : Real := 8.0;   // kW
   END_VAR
BEGIN

REGION Network 1 (SCL)
   // Inverters. Do not convert to ELSIF
   IF "DB_InverterDrives".CPC_SC_01.Stat.Power.Eng.bError = FALSE THEN
       #fPower += "DB_InverterDrives".CPC_SC_01.Stat.Power.Eng.fValue;
   END_IF;
   IF "DB_InverterDrives".HBL_SC_01.Stat.Power.Eng.bError = FALSE THEN
       #fPower += "DB_InverterDrives".HBL_SC_01.Stat.Power.Eng.fValue;
   END_IF;
   IF "DB_InverterDrives".HBL_SC_02.Stat.Power.Eng.bError = FALSE THEN
       #fPower += "DB_InverterDrives".HBL_SC_02.Stat.Power.Eng.fValue;
   END_IF;
   IF "DB_InverterDrives".HBL_SC_10.Stat.Power.Eng.bError = FALSE THEN
       #fPower += "DB_InverterDrives".HBL_SC_10.Stat.Power.Eng.fValue;
   END_IF;

   // Auxiliary Motors. Do not convert to ELSIF
   IF "DB_DO".SSC_P_01 = TRUE THEN
       #fPower += #SSC_P_01_POWER;
   END_IF;
   IF "DB_DO".SSC_P_02 = TRUE THEN
       #fPower += #SSC_P_02_POWER;
   END_IF;
   IF "DB_DO".SSC_F_01 = TRUE THEN
       #fPower += #SSC_F_01_POWER;
   END_IF;
   IF "DB_DO".CPC_P_01 = TRUE THEN
       #fPower += #CPC_P_01_POWER;
   END_IF;

   // Cabinet heating & cooling. Do not convert to ELSIF
   IF "DB_DO".CabinetHeater = TRUE THEN
       #fPower += #CabinetHeater_POWER;
   END_IF;
   IF "DB_DO".CabinetFan = TRUE THEN
       #fPower += #CabinetHeater_POWER;
   END_IF;

   // Crankcase oil heaters. Do not convert to ELSIF
   IF "DB_DO".HBL_EC_01 = TRUE THEN
       #fPower += #HBL_EC_01_POWER;
   END_IF;
   IF "DB_DO".HBL_EC_02 = TRUE THEN
       #fPower += #HBL_EC_02_POWER;
   END_IF;

   // Store in calc object
   "fcCalcAssign"(fValue := #fPower, sTag := "DB_Calc".System.ElectricalPower);
END_REGION
END_FUNCTION

FUNCTION "DT1" : Real
{ S7_Optimized_Access := 'TRUE' }
VERSION : 0.1
   VAR_INPUT 
      u : Real;
      T1 : Real;
      fCycleTime : Real;
   END_VAR

   VAR_IN_OUT 
      xh_merk : Real;
   END_VAR

   VAR_TEMP 
      tt1 : Real;
      Du : Real;
   END_VAR


BEGIN
	// These is a discrete filtered derivative function. With the filter time T.
	// With a constant increasing/decreasing value u the output y is the change rate per second.
	// the step response is a decreasing exponential function that is proportional to the step size and almost zero (<1%) after 5*T. The surface (integral) over it is the step size from the input function.
	// if the filter time T is zero, it’s an ideal descref integral (u-u_old)/cycle time
	
	//Reset if xh_merk is NaN
	IF "isNaN"(#xh_merk ) THEN 
	    #xh_merk := #u; 
	END_IF;
	
	#DT1 := (#u - #xh_merk) / (#T1 + #fCycleTime);
	#xh_merk := #xh_merk + #fCycleTime * #DT1;
END_FUNCTION

FUNCTION_BLOCK "OperatingTimeCounters"   // FB41, FBD
{ S7_Optimized_Access := 'TRUE' }
VERSION : 0.1
// stored: AutoNumber true, IsIECCheckEnabled false, IsRetainMemResEnabled false, MemoryReserve 0, SetENOAutomatically false, UDAEnableTagReadback false
   VAR
      SystemOnTime { ExternalAccessible := 'False'; ExternalVisible := 'False'; ExternalWritable := 'False'} : "fbHoursCounter";
      SwitchedOnTime { ExternalAccessible := 'False'; ExternalVisible := 'False'; ExternalWritable := 'False'; S7_SetPoint := 'True'} : "fbHoursCounter";
      RunningTime { ExternalAccessible := 'False'; ExternalVisible := 'False'; ExternalWritable := 'False'; S7_SetPoint := 'True'} : "fbHoursCounter";
      RuntimeMemory { ExternalAccessible := 'False'; ExternalVisible := 'False'; ExternalWritable := 'False'; S7_SetPoint := 'True'} : LReal;
   END_VAR
BEGIN

REGION Network 1: Read out scan time
   // This is in the wrong place
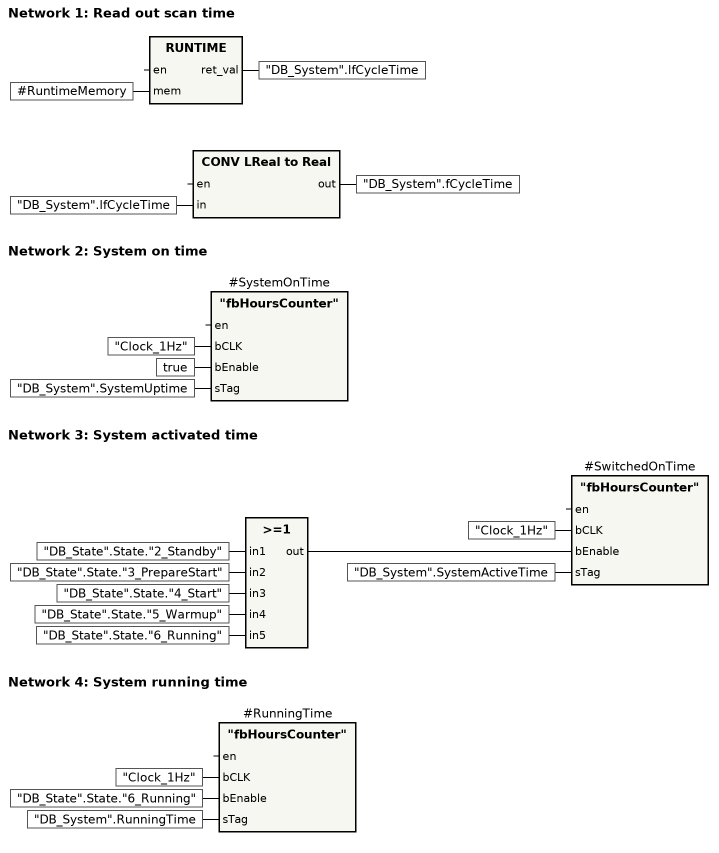
   // no SCL statement known for Runtime: written as a call
   "DB_System".lfCycleTime := Runtime(mem := #RuntimeMemory);
   "DB_System".fCycleTime := LREAL_TO_REAL("DB_System".lfCycleTime);
END_REGION

REGION Network 2: System on time
   #SystemOnTime(bCLK := "Clock_1Hz", bEnable := true, sTag := "DB_System".SystemUptime);   // "fbHoursCounter"
END_REGION

REGION Network 3: System activated time
   #SwitchedOnTime(bCLK := "Clock_1Hz",   // "fbHoursCounter"
                   bEnable := "DB_State".State."2_Standby" OR "DB_State".State."3_PrepareStart" OR "DB_State".State."4_Start" OR "DB_State".State."5_Warmup" OR "DB_State".State."6_Running",
                   sTag := "DB_System".SystemActiveTime);
END_REGION

REGION Network 4: System running time
   #RunningTime(bCLK := "Clock_1Hz", bEnable := "DB_State".State."6_Running", sTag := "DB_System".RunningTime);   // "fbHoursCounter"
END_REGION
END_FUNCTION_BLOCK

FUNCTION_BLOCK "fbHoursCounter"   // FB36, FBD
TITLE = Hours counter
{ S7_Optimized_Access := 'TRUE' }
VERSION : 0.1
// When Enable = TRUE, increase the elapsed time count
// stored: AutoNumber true, IsIECCheckEnabled false, IsRetainMemResEnabled false, MemoryReserve 0, SetENOAutomatically false, UDAEnableTagReadback false
   VAR_INPUT
      bCLK : Bool;   // 1-second pulse
      bEnable : Bool;   // Enable counting
   END_VAR
   VAR_IN_OUT
      sTag : "stHoursCounter";
   END_VAR
   VAR RETAIN
      Hours : CTU_UDINT;
      Minutes { S7_SetPoint := 'True'} : CTU_USINT;
      Seconds { S7_SetPoint := 'True'} : CTU_USINT;
   END_VAR
   VAR
      Rollover_sec { S7_SetPoint := 'True'} : Bool;
      Rollover_min : Bool;
   END_VAR
   VAR_TEMP
      Clock : Bool;
   END_VAR
BEGIN

REGION Network 1: Gate clock bit
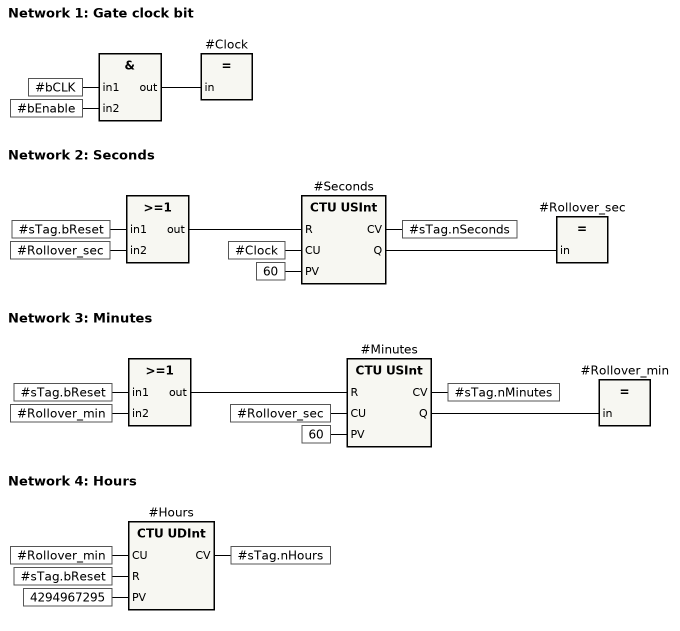
   #Clock := #bCLK AND #bEnable;
END_REGION

REGION Network 2: Seconds
   #Seconds(R := #sTag.bReset OR #Rollover_sec, CU := #Clock, PV := 60, CV => #sTag.nSeconds);   // CTU
   #Rollover_sec := #Seconds.Q;
END_REGION

REGION Network 3: Minutes
   #Minutes(R := #sTag.bReset OR #Rollover_min, CU := #Rollover_sec, PV := 60, CV => #sTag.nMinutes);   // CTU
   #Rollover_min := #Minutes.Q;
END_REGION

REGION Network 4: Hours
   // Note: this is not automatically reset, should count up "forever" (approx equal to 490293 years).
   #Hours(CU := #Rollover_min, R := #sTag.bReset, PV := 4294967295, CV => #sTag.nHours);   // CTU
END_REGION
END_FUNCTION_BLOCK

FUNCTION_BLOCK "StateMachine"   // FB4, FBD
TITLE = Handling of machine states
{ S7_Optimized_Access := 'TRUE' }
VERSION : 0.1
// NB: the bit for each state stays high for one cycle after leaving the state. So when leaving State 2 for State 3, on the first cycle #StateChanges."2-zu-3_StateChange" will go high, setting the State 3 bit. But since the reset of State 2 is in an earlier network, this can't happen until the next cycle. So #StateChanges."2-zu-3_StateChange" has to stay high for the second cycle, when it causes State 2 RS to be reset. On the third cycle then also #StateChanges."2-zu-3_StateChange" is FALSE due to the State. This is subtle and tricky behaviour, not the best, rewrite this one day
// stored: AutoNumber true, IsIECCheckEnabled false, IsRetainMemResEnabled false, MemoryReserve 0, SetENOAutomatically false, UDAEnableTagReadback false
   VAR
      StateChanges : Struct
         "0-zu-1_StateChange" : Bool;
         "1-zu-2_StateChange" : Bool;
         "2-zu-3_StateChange" : Bool;
         "2-zu-7_StateChange" : Bool;
         "3-zu-2_StateChange" : Bool;
         "3-zu-4_StateChange" : Bool;
         "3-zu-7_StateChange" : Bool;
         "4-zu-2_StateChange" : Bool;
         "4-zu-5_StateChange" : Bool;
         "4-zu-7_StateChange" : Bool;
         "5-zu-2_StateChange" : Bool;
         "5-zu-6_StateChange" : Bool;
         "5-zu-7_StateChange" : Bool;
         "6-zu-2_StateChange" : Bool;
         "6-zu-7_StateChange" : Bool;
         "7-zu-1_StateChange" : Bool;
      END_STRUCT;
      Evaluate_DB : "Evaluate";
   END_VAR
   VAR_TEMP   // added for the SCL form of the ladder/FBD networks
      _w1 : Bool;
   END_VAR
BEGIN

REGION Network 1: Evaluate machine conditions
